ABB RAPID module: FOUNDRY.mod

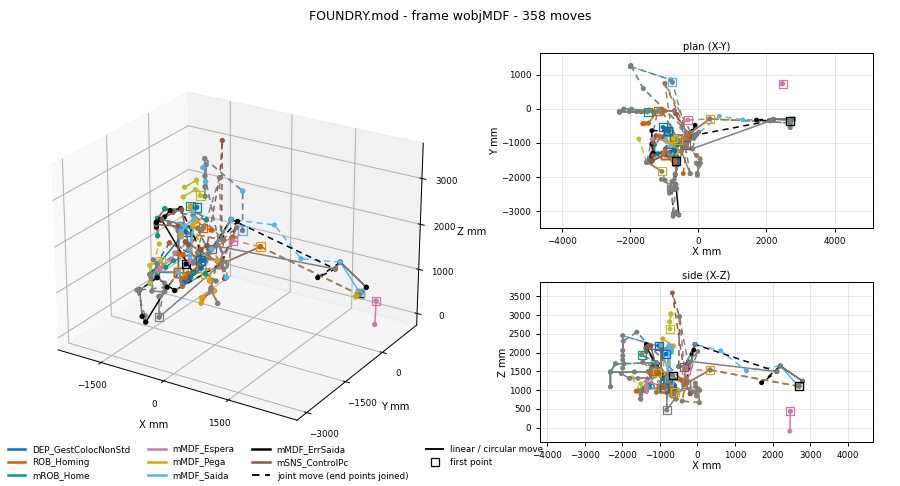
[picture p0: tool path of FOUNDRY.mod in frame wobjMDF, 358 of 371 moves have a stored position in this frame; points joined in program order, loops and branches not executed]
MODULE FOUNDRY

    !***********************************************************************************
    !*Project:   customer			: CIE Autocom (BR)
    !*           robot s/n			: 8156
    !*
    !*Robot:     Robot System		: IRC5 6.04.01.00
    !*           Robot NR.			: 109474
    !*           Robot Option		:
    !*           Robot Type			: IRB 6700-205/2.80
    !*           Robot Software		:
    !*           TP Language		: PORTUGUES
    !*
    !*Periferie: DCM type			: COLOSIO PFO2000
    !*           cooling device		: vasca (cliente)
    !*           photosensors		: SI (Ligado ao conrolador do robô)
    !*           conveyor belt		: SI
    !*           spraying			: NO
    !*           trimming press		: SI (collegata a controller robot)I
    !*
    !*Created:	 2017-02-17
    !*Author:    A.Roberti
    !*Company:   RELBO srl
    !*Modified:  Fabio Luiz dos Santos
    !*Translated to portuguese: Fabio Luiz dos Santos
    !*
    !*THIS MODULE MUST BE USED WITH "TEXT", "UTILITY" AND "WLDZONES" MODULES.
    !***********************************************************************************

    !============ Conferir posições abaixo ============
    CONST robtarget p01:=[[2473.51,738.92,438.42],[0.454099,0.457405,0.552238,0.528779],[1,0,0,1],[9E+09,9E+09,9E+09,9E+09,9E+09,9E+09]];
    CONST robtarget p02:=[[2460.24,732.08,-92.92],[0.449187,0.452046,0.556362,0.533242],[1,0,0,1],[9E+09,9E+09,9E+09,9E+09,9E+09,9E+09]];
    PERS robtarget pTemp:=[[2468.78,703.01,-92.8363],[0.452338,0.45528,0.553646,0.530647],[1,0,0,1],[9E+09,9E+09,9E+09,9E+09,9E+09,9E+09]];
    CONST robtarget p04:=[[2373.93,-299.91,1461.99],[0.596392,-6.67991E-05,0.802693,-2.09958E-05],[1,-1,-1,1],[9E+09,9E+09,9E+09,9E+09,9E+09,9E+09]];
    CONST robtarget p05:=[[2373.93,-299.91,1461.99],[0.596392,-6.67991E-05,0.802693,-2.09958E-05],[1,-1,-1,1],[9E+09,9E+09,9E+09,9E+09,9E+09,9E+09]];
    CONST robtarget p06:=[[2373.93,-299.91,1461.99],[0.596392,-6.67991E-05,0.802693,-2.09958E-05],[1,-1,-1,1],[9E+09,9E+09,9E+09,9E+09,9E+09,9E+09]];
    CONST robtarget MDF_pRecog10:=[[2695.82,-242.69,1199.03],[0.998237,-0.00496931,0.0559359,-0.0192193],[1,-1,-1,1],[9E+09,9E+09,9E+09,9E+09,9E+09,9E+09]];

    CONST robtarget MDF_p23:=[[-309.29,-759.88,1174.58],[0.243259,-0.675086,-0.655856,-0.234385],[0,-1,0,0],[9E+09,9E+09,9E+09,9E+09,9E+09,9E+09]];
    CONST robtarget MDF_p41:=[[2057.65,-246.89,1441.09],[0.616132,-0.00865147,0.787526,0.0104616],[1,-1,0,1],[9E+09,9E+09,9E+09,9E+09,9E+09,9E+09]];
    CONST robtarget MDF_p40:=[[1706.22,-328.45,1196.02],[0.687339,-0.0878871,0.720939,-0.00939877],[1,-1,-1,1],[9E+09,9E+09,9E+09,9E+09,9E+09,9E+09]];
    CONST robtarget MDF_p51:=[[2695.80,-284.56,1199.03],[0.998236,-0.0049758,0.0559417,-0.0192583],[1,-1,-1,1],[9E+09,9E+09,9E+09,9E+09,9E+09,9E+09]];
    CONST robtarget MDF_p50:=[[2695.80,-284.56,1199.03],[0.998236,-0.00497575,0.0559413,-0.0192576],[1,-1,-1,1],[9E+09,9E+09,9E+09,9E+09,9E+09,9E+09]];
    CONST robtarget MDF_p60:=[[2695.80,-284.56,1199.03],[0.998236,-0.00497576,0.0559417,-0.0192575],[1,-1,-1,1],[9E+09,9E+09,9E+09,9E+09,9E+09,9E+09]];
    CONST robtarget MDF_p61:=[[2695.80,-284.56,1199.03],[0.998236,-0.00497571,0.0559408,-0.0192572],[1,-1,-1,1],[9E+09,9E+09,9E+09,9E+09,9E+09,9E+09]];
    CONST robtarget MDF_p22:=[[1102.79,-218.74,1895.07],[0.935496,-0.0143034,0.351181,0.036262],[1,-1,0,1],[9E+09,9E+09,9E+09,9E+09,9E+09,9E+09]];

    CONST robtarget MDF_p70:=[[93.40,-478.70,2065.31],[0.934668,0.0189998,0.0567069,-0.350456],[1,-1,0,1],[9E+09,9E+09,9E+09,9E+09,9E+09,9E+09]];
    CONST robtarget MDF_p71:=[[-94.08,-478.58,2065.27],[0.849875,0.0295531,0.0520109,-0.523578],[0,-1,0,1],[9E+09,9E+09,9E+09,9E+09,9E+09,9E+09]];
    CONST robtarget MDF_p80:=[[1370.80,-212.89,1499.22],[0.814032,-0.0190361,0.57994,0.0256936],[1,-1,-1,1],[9E+09,9E+09,9E+09,9E+09,9E+09,9E+09]];
    CONST robtarget MDF_p81:=[[1306.48,-320.84,1511.93],[0.617506,-0.130992,0.771355,0.0808671],[1,-1,0,1],[9E+09,9E+09,9E+09,9E+09,9E+09,9E+09]];

    CONST robtarget MDF_p91:=[[617.59,-214.31,2051.16],[0.805845,-0.0646225,-0.0933712,0.581137],[1,0,0,1],[9E+09,9E+09,9E+09,9E+09,9E+09,9E+09]];
    CONST robtarget MDF_p33:=[[319.27,-312.34,1536.54],[0.13049,0.0260758,0.991098,-0.00401919],[1,-1,0,0],[9E+09,9E+09,9E+09,9E+09,9E+09,9E+09]];
    CONST robtarget MDF_pControl10:=[[448.88,-592.67,2016.31],[0.996524,0.0429781,0.0652434,-0.0289314],[1,0,0,1],[9E+09,9E+09,9E+09,9E+09,9E+09,9E+09]];
    CONST robtarget MDF_p43:=[[2697.36,-501.35,1107.86],[0.998235,-0.00496071,0.055963,-0.0192532],[1,-1,0,1],[9E+09,9E+09,9E+09,9E+09,9E+09,9E+09]];
    CONST robtarget MDF_p32:=[[-148.76,-493.05,1985.25],[0.747821,0.0411262,0.131836,-0.649378],[0,-1,-1,1],[9E+09,9E+09,9E+09,9E+09,9E+09,9E+09]];
    CONST robtarget SNS_p21:=[[-309.29,-759.88,1174.58],[0.243257,-0.67509,-0.655856,-0.234378],[0,-1,0,0],[9E+09,9E+09,9E+09,9E+09,9E+09,9E+09]];
    CONST robtarget pControl_01:=[[-304.77,-1154.52,1895.14],[0.698253,-0.00430576,0.705523,-0.121086],[0,-2,0,1],[9E+09,9E+09,9E+09,9E+09,9E+09,9E+09]];


    !===================================================================================
    ! EIXOS EM 0 GRAUS PARA VERIFICAR CALIBRACAO
    CONST jointtarget jposCalib:=[[0.0,0.0,0.0,0.0,0.0,0.0],[9E+09,9E+09,9E+09,9E+09,9E+09,9E+09]];
    ! POSICAO DE TRANSPORTE
    CONST jointtarget jposTransporte:=[[0.00449267,-45.002,64.9985,0.000647968,-115.001,4.99587],[9E+09,9E+09,9E+09,9E+09,9E+09,9E+09]];
    !===================================================================================
    ! HOME POSICAO (POSICAO INICIAL)
    CONST robtarget ROB_pHome:=[[-309.29,-759.88,1174.59],[0.243259,-0.67509,-0.655854,-0.23438],[0,-1,0,0],[9E+09,9E+09,9E+09,9E+09,9E+09,9E+09]];
    !===================================================================================
    ! M?QUINA DE FUNDICAO (MDF): ESPERA
    CONST robtarget MDF_pEspera:=[[335.19,-295.19,1536.55],[0.13056,9.64202E-05,0.99144,-0.00060735],[1,-1,0,0],[9E+09,9E+09,9E+09,9E+09,9E+09,9E+09]];
    !===================================================================================
    ! MAQUINA DE FUNDICAO (MDF): ENTRADA
    CONST robtarget MDF_p01:=[[2704.71,-411.78,1100.79],[0.587037,0.011242,0.809463,0.00555487],[1,-1,0,1],[9E+09,9E+09,9E+09,9E+09,9E+09,9E+09]];
    CONST robtarget MDF_p02:=[[2697.36,-357.61,1107.87],[0.998235,-0.00496108,0.0559633,-0.0192572],[1,-1,-1,1],[9E+09,9E+09,9E+09,9E+09,9E+09,9E+09]];
    CONST robtarget MDF_p03:=[[2697.37,-358.92,1107.86],[0.998235,-0.00495896,0.0559656,-0.0192394],[1,-1,-1,1],[9E+09,9E+09,9E+09,9E+09,9E+09,9E+09]];
    CONST robtarget MDF_pPega:=[[2697.36,-549.12,1107.87],[0.998235,-0.00496031,0.055963,-0.0192579],[1,-1,0,1],[9E+09,9E+09,9E+09,9E+09,9E+09,9E+09]];
    PERS robtarget MDF_pTemp:=[[2694.21,-536.375,1106.5],[0.998116,-0.00503237,0.0568545,-0.0225023],[1,-1,0,1],[9E+09,9E+09,9E+09,9E+09,9E+09,9E+09]];
    CONST robtarget MDF_p04:=[[2697.36,-297.72,1107.87],[0.998235,-0.00496111,0.0559628,-0.019259],[1,-1,-1,1],[9E+09,9E+09,9E+09,9E+09,9E+09,9E+09]];
    !===================================================================================
    ! MAQUINA DE FUNDICAO (MDF): SALIDA
    CONST robtarget MDF_p10:=[[2798.70,-298.15,1239.60],[0.868299,-0.0143122,0.495492,-0.0184121],[1,-1,-1,1],[9E+09,9E+09,9E+09,9E+09,9E+09,9E+09]];
    CONST robtarget MDF_p11:=[[2203.10,-303.56,1644.90],[0.856797,-0.177507,0.433581,0.215401],[1,-1,0,1],[9E+09,9E+09,9E+09,9E+09,9E+09,9E+09]];
    CONST robtarget MDF_p12:=[[2114.45,-349.91,1492.71],[0.599346,-0.117299,0.78976,0.0574839],[1,-1,0,1],[9E+09,9E+09,9E+09,9E+09,9E+09,9E+09]];
    CONST robtarget MDF_p20:=[[1642.01,-439.61,1289.54],[0.823576,-5.9409E-05,0.567206,-1.43407E-05],[1,-1,0,1],[9E+09,9E+09,9E+09,9E+09,9E+09,9E+09]];
    CONST robtarget MDF_p21:=[[992.58,-330.88,1566.27],[0.702618,-0.0208979,0.710504,-0.0327757],[1,-1,0,1],[9E+09,9E+09,9E+09,9E+09,9E+09,9E+09]];
    CONST robtarget MDF_pControl:=[[-165.98,-1166.57,1763.98],[0.60515,0.0268408,0.791448,-0.0817503],[0,-2,0,1],[9E+09,9E+09,9E+09,9E+09,9E+09,9E+09]];
    CONST robtarget MDF_pControl_11:=[[-304.77,-1154.52,1895.14],[0.698253,-0.00430576,0.705523,-0.121086],[0,-2,0,1],[9E+09,9E+09,9E+09,9E+09,9E+09,9E+09]];
    CONST robtarget MDF_p30:=[[-66.69,-765.21,2217.81],[0.991581,-0.108659,-0.0385252,-0.0589544],[0,0,0,1],[9E+09,9E+09,9E+09,9E+09,9E+09,9E+09]];
    CONST robtarget MDF_p31:=[[-350.61,-1056.76,1612.90],[0.680926,0.0158107,0.727045,-0.0865753],[-1,-2,0,1],[9E+09,9E+09,9E+09,9E+09,9E+09,9E+09]];
    CONST robtarget MDF_p13:=[[-309.29,-759.89,1174.59],[0.243258,-0.67509,-0.655855,-0.23438],[0,-1,0,0],[9E+09,9E+09,9E+09,9E+09,9E+09,9E+09]];
    CONST robtarget MDF_p14:=[[12.02,-682.53,2028.46],[0.998079,0.0593523,0.0134589,-0.0115613],[0,-1,0,1],[9E+09,9E+09,9E+09,9E+09,9E+09,9E+09]];
    !===================================================================================
    ! SENSORES
    CONST robtarget SNS_p01:=[[-350.61,-1056.76,1612.89],[0.680927,0.0158161,0.727044,-0.0865756],[-1,-2,0,1],[9E+09,9E+09,9E+09,9E+09,9E+09,9E+09]];
    CONST robtarget SNS_p02:=[[-498.09,-998.45,1630.02],[0.680911,0.0157817,0.727055,-0.086622],[-1,-2,0,1],[9E+09,9E+09,9E+09,9E+09,9E+09,9E+09]];
    CONST robtarget SNS_pControl1:=[[-498.07,-1238.79,1630.02],[0.680913,0.0157813,0.727053,-0.0866156],[-1,-2,0,1],[9E+09,9E+09,9E+09,9E+09,9E+09,9E+09]];
    CONST robtarget SNS_pControl2:=[[-236.59,-1901.29,1658.69],[0.555085,0.419469,-0.460857,0.550942],[0,1,0,0],[9E+09,9E+09,9E+09,9E+09,9E+09,9E+09]];
    CONST robtarget SNS_pControl3:=[[-236.59,-1901.29,1658.69],[0.555086,0.419469,-0.460856,0.550942],[0,1,0,0],[9E+09,9E+09,9E+09,9E+09,9E+09,9E+09]];
    CONST robtarget SNS_pControl4:=[[-236.59,-1901.29,1658.69],[0.555085,0.419469,-0.460857,0.550942],[0,1,0,0],[9E+09,9E+09,9E+09,9E+09,9E+09,9E+09]];
    CONST robtarget SNS_p10:=[[-479.84,-542.93,2956.94],[0.0253695,-0.0230724,0.928121,-0.370697],[-1,-2,0,1],[9E+09,9E+09,9E+09,9E+09,9E+09,9E+09]];
    CONST robtarget SNS_p11:=[[-309.29,-759.88,1174.59],[0.24326,-0.67509,-0.655854,-0.234381],[0,-1,0,0],[9E+09,9E+09,9E+09,9E+09,9E+09,9E+09]];
    !=====================================================================================
    ! CUBA DE AGUA
    CONST robtarget ENF_p01:=[[-816.23,-2285.86,928.08],[0.215617,0.952924,0.0580622,0.205121],[0,0,0,0],[9E+09,9E+09,9E+09,9E+09,9E+09,9E+09]];
    CONST robtarget ENF_p02:=[[-440.63,-1897.38,1282.18],[0.718138,0.0885909,0.689911,-0.0212891],[0,-2,0,1],[9E+09,9E+09,9E+09,9E+09,9E+09,9E+09]];
    CONST robtarget ENF_p03:=[[-573.40,-2628.84,1240.28],[0.718462,0.0885711,0.689567,-0.0215669],[0,-2,0,1],[9E+09,9E+09,9E+09,9E+09,9E+09,9E+09]];
    CONST robtarget ENF_p04:=[[-785.25,-1953.16,845.96],[0.631902,0.761096,0.0876551,0.11726],[0,1,-1,0],[9E+09,9E+09,9E+09,9E+09,9E+09,9E+09]];
    CONST robtarget ENF_pCuba:=[[-816.30,-2285.83,472.77],[0.215579,0.952925,0.0580234,0.205164],[0,0,0,0],[9E+09,9E+09,9E+09,9E+09,9E+09,9E+09]];
    CONST robtarget ENF_p10:=[[-778.88,-2131.13,1173.74],[0.71674,0.696411,0.000326903,-0.0360001],[0,1,-1,0],[9E+09,9E+09,9E+09,9E+09,9E+09,9E+09]];
    CONST robtarget ENF_p11:=[[-780.71,-2290.62,948.87],[0.631901,0.761095,0.0876729,0.117254],[0,1,-1,0],[9E+09,9E+09,9E+09,9E+09,9E+09,9E+09]];
    CONST robtarget ENF_p12:=[[29.47,-1884.57,501.58],[0.106643,-0.639134,-0.750945,0.127342],[0,-3,2,1],[9E+09,9E+09,9E+09,9E+09,9E+09,9E+09]];
    CONST robtarget ENF_p20:=[[-633.19,-2343.32,1104.45],[0.431426,0.658438,-0.391718,0.476328],[0,1,0,0],[9E+09,9E+09,9E+09,9E+09,9E+09,9E+09]];
    CONST robtarget ENF_p21:=[[-1085.76,-2068.67,1587.93],[0.646248,0.686559,0.136448,-0.303944],[0,1,-2,0],[9E+09,9E+09,9E+09,9E+09,9E+09,9E+09]];
    CONST robtarget ENF_p22:=[[-972.77,-2097.81,1535.68],[0.696167,0.699868,-0.0129623,-0.159272],[0,1,-1,0],[9E+09,9E+09,9E+09,9E+09,9E+09,9E+09]];
    CONST robtarget ENF_p23:=[[-440.54,-1897.37,1282.17],[0.718139,0.0885822,0.689911,-0.0212782],[0,-2,0,1],[9E+09,9E+09,9E+09,9E+09,9E+09,9E+09]];
    !===================================================================================
    ! COLOCACAO PECA NO INTERMEDIARIO
    CONST robtarget UTL_p01:=[[-1070.06,-1835.10,1470.49],[0.466574,0.842745,-0.106745,-0.246362],[0,1,-1,1],[9E+09,9E+09,9E+09,9E+09,9E+09,9E+09]];
    CONST robtarget UTL_p02:=[[-1293.78,-1608.42,1558.93],[0.831149,0.370293,-0.213137,-0.355874],[0,0,0,1],[9E+09,9E+09,9E+09,9E+09,9E+09,9E+09]];
    CONST robtarget UTL_p03:=[[-1482.11,-1589.62,1388.74],[0.54708,0.552185,-0.433217,-0.456201],[0,0,0,1],[9E+09,9E+09,9E+09,9E+09,9E+09,9E+09]];
    CONST robtarget UTL_p04:=[[-1505.03,-1545.60,877.79],[0.493718,0.499244,-0.496928,-0.509962],[0,0,0,1],[9E+09,9E+09,9E+09,9E+09,9E+09,9E+09]];
    CONST robtarget UTL_pColoc:=[[-1509.62,-1576.07,771.05],[0.59829,0.613623,-0.36049,-0.368189],[0,0,0,1],[9E+09,9E+09,9E+09,9E+09,9E+09,9E+09]];
    CONST robtarget UTL_p10:=[[-1504.86,-1545.34,953.20],[0.493701,0.499248,-0.496933,-0.509969],[0,0,0,1],[9E+09,9E+09,9E+09,9E+09,9E+09,9E+09]];
    CONST robtarget UTL_p11:=[[-1742.50,-882.65,1329.94],[0.547038,0.552222,-0.433233,-0.45619],[-1,0,0,1],[9E+09,9E+09,9E+09,9E+09,9E+09,9E+09]];
    CONST robtarget UTL_p12:=[[-1479.96,-1594.74,1007.69],[0.547037,0.552216,-0.433221,-0.45621],[0,0,0,1],[9E+09,9E+09,9E+09,9E+09,9E+09,9E+09]];
    !===================================================================================
    ! RETIRADA PECA DO INTERMEDIARIO
    CONST robtarget UTL_p51:=[[-837.41,-1272.63,1959.31],[0.955925,0.0359635,-0.0135944,-0.291083],[0,0,0,1],[9E+09,9E+09,9E+09,9E+09,9E+09,9E+09]];
    CONST robtarget UTL_p52:=[[-1296.42,-1371.93,1145.58],[0.695048,0.651142,0.261802,0.156151],[-1,-2,1,1],[9E+09,9E+09,9E+09,9E+09,9E+09,9E+09]];
    CONST robtarget UTL_p53:=[[-1296.41,-1372.01,1145.58],[0.695055,0.651133,0.261809,0.156144],[-1,-2,1,1],[9E+09,9E+09,9E+09,9E+09,9E+09,9E+09]];
    CONST robtarget UTL_p54:=[[-1505.01,-1545.57,877.73],[0.493703,0.499257,-0.496926,-0.509965],[0,0,0,1],[9E+09,9E+09,9E+09,9E+09,9E+09,9E+09]];
    CONST robtarget UTL_pPega:=[[-1510.35,-1566.50,762.25],[0.502673,0.515186,-0.488253,-0.49347],[0,0,0,1],[9E+09,9E+09,9E+09,9E+09,9E+09,9E+09]];
    CONST robtarget UTL_p60:=[[-1504.87,-1545.36,953.30],[0.493713,0.499235,-0.496941,-0.509963],[0,0,0,1],[9E+09,9E+09,9E+09,9E+09,9E+09,9E+09]];
    CONST robtarget UTL_p61:=[[-1434.58,-1608.11,1694.89],[0.663,0.645996,-0.264879,-0.270111],[0,0,0,1],[9E+09,9E+09,9E+09,9E+09,9E+09,9E+09]];
    CONST robtarget UTL_p62:=[[-1196.41,-1319.01,1646.77],[0.655082,0.649295,-0.283991,-0.261979],[0,0,0,1],[9E+09,9E+09,9E+09,9E+09,9E+09,9E+09]];
    !===================================================================================
    ! PRENSA: COLOCACAO
    CONST robtarget PRN_p01:=[[-1193.80,-61.32,1513.33],[0.15952,0.928352,-0.262292,-0.20957],[-1,0,0,0],[9E+09,9E+09,9E+09,9E+09,9E+09,9E+09]];
    CONST robtarget PRN_p02:=[[-976.84,-61.28,1510.97],[0.233234,0.684208,-0.682248,-0.109542],[-1,0,0,0],[9E+09,9E+09,9E+09,9E+09,9E+09,9E+09]];
    CONST robtarget PRN_p03:=[[-1453.00,-37.75,1743.34],[0.498689,0.512749,-0.4968,-0.491515],[-1,0,0,1],[9E+09,9E+09,9E+09,9E+09,9E+09,9E+09]];
    CONST robtarget PRN_p04:=[[-2008.40,-78.87,1584.76],[0.505059,0.503661,-0.494129,-0.497069],[-1,0,0,1],[9E+09,9E+09,9E+09,9E+09,9E+09,9E+09]];
    CONST robtarget PRN_p05:=[[-2025.32,-80.39,1437.60],[0.519828,0.551911,-0.473982,-0.447788],[-1,-1,1,1],[9E+09,9E+09,9E+09,9E+09,9E+09,9E+09]];
    CONST robtarget PRN_p06:=[[-2012.84,-78.16,1221.12],[0.519832,0.551906,-0.47397,-0.447802],[-1,-1,1,1],[9E+09,9E+09,9E+09,9E+09,9E+09,9E+09]];
    PERS robtarget PRN_pColoc:=[[-2031.56,-75.53,1091.03],[0.510214,0.51944,-0.489066,-0.480291],[-1,-1,1,1],[9E+09,9E+09,9E+09,9E+09,9E+09,9E+09]];
    CONST robtarget PRN_p10:=[[-2025.32,-80.42,1437.60],[0.519832,0.551912,-0.473979,-0.447785],[-1,-1,1,1],[9E+09,9E+09,9E+09,9E+09,9E+09,9E+09]];
    CONST robtarget PRN_p11:=[[-1804.46,-79.94,1313.09],[0.501985,0.498001,-0.498114,-0.501885],[-1,0,0,1],[9E+09,9E+09,9E+09,9E+09,9E+09,9E+09]];
    CONST robtarget PRN_p12:=[[-1586.23,-73.82,1311.37],[0.501982,0.498008,-0.49812,-0.501876],[-1,0,0,1],[9E+09,9E+09,9E+09,9E+09,9E+09,9E+09]];
    CONST robtarget PRN_p13:=[[-695.62,-55.45,1352.81],[0.0390151,0.751501,-0.655563,0.0629308],[-1,0,0,0],[9E+09,9E+09,9E+09,9E+09,9E+09,9E+09]];
    CONST robtarget PRN_p14:=[[-695.62,-55.41,1352.84],[0.0390281,0.751508,-0.655556,0.0629139],[-1,0,0,0],[9E+09,9E+09,9E+09,9E+09,9E+09,9E+09]];
    !
    !   Posicoes de deposito na prensa dependentes de retirada da gaveta
    !
    PERS robtarget pDepositaPrensa_1:=[[-2031.56,-75.53,1091.03],[0.510214,0.51944,-0.489066,-0.480291],[-1,-1,1,1],[9E+09,9E+09,9E+09,9E+09,9E+09,9E+09]];
    PERS robtarget pDepositaPrensa_2:=[[-2025.94,-80.41,1132.31],[0.508364,0.51283,-0.495652,-0.482598],[-1,-1,1,1],[9E+09,9E+09,9E+09,9E+09,9E+09,9E+09]];
    PERS robtarget pDepositaPrensa_3:=[[-2032.75,-74.5,1096.36],[0.511914,0.521062,-0.487274,-0.478543],[-1,-1,1,1],[9E+09,9E+09,9E+09,9E+09,9E+09,9E+09]];
    PERS robtarget pDepositaPrensa_4:=[[-2029.34,-74.63,1090.39],[0.513337,0.522498,-0.485777,-0.476972],[-1,-1,1,1],[9E+09,9E+09,9E+09,9E+09,9E+09,9E+09]];
    PERS robtarget pDepositaPrensa_5:=[[-2022.17,-74.64,1099.64],[0.497093,0.506578,-0.50237,-0.493864],[-1,0,0,1],[9E+09,9E+09,9E+09,9E+09,9E+09,9E+09]];
    PERS robtarget pDepositaPrensa_6:=[[-2022.17,-74.64,1099.64],[0.497093,0.506578,-0.50237,-0.493864],[-1,0,0,1],[9E+09,9E+09,9E+09,9E+09,9E+09,9E+09]];
    !
    !===================================================================================
    ! PRENSA: RETIRADA
    CONST robtarget PRN_p50:=[[-1486.38,-85.78,1945.73],[0.0614075,-0.701391,-0.688555,0.173702],[-1,0,3,0],[9E+09,9E+09,9E+09,9E+09,9E+09,9E+09]];
    CONST robtarget PRN_p51:=[[-1089.99,-98.97,1732.92],[0.222555,0.667241,0.697434,0.137275],[-1,0,3,0],[9E+09,9E+09,9E+09,9E+09,9E+09,9E+09]];
    CONST robtarget PRN_p52:=[[-1959.35,-6.29,1703.73],[0.497499,-0.502459,-0.49938,0.500649],[-1,0,3,1],[9E+09,9E+09,9E+09,9E+09,9E+09,9E+09]];
    CONST robtarget PRN_p53:=[[-2182.85,-6.28,1702.88],[0.497495,-0.502467,-0.499382,0.500642],[-1,0,3,1],[9E+09,9E+09,9E+09,9E+09,9E+09,9E+09]];
    CONST robtarget PRN_p54:=[[-2317.52,-87.25,1480.78],[0.497056,-0.502836,-0.499704,0.500388],[-1,0,2,1],[9E+09,9E+09,9E+09,9E+09,9E+09,9E+09]];
    CONST robtarget PRN_pPega:=[[-2315.98,-96.83,1089.21],[0.490704,-0.516807,-0.502931,0.489061],[-1,0,2,1],[9E+09,9E+09,9E+09,9E+09,9E+09,9E+09]];
    CONST robtarget PRN_p60:=[[-2317.51,-87.34,1480.84],[0.497055,-0.502826,-0.499706,0.500396],[-1,0,2,1],[9E+09,9E+09,9E+09,9E+09,9E+09,9E+09]];
    PERS robtarget PRN_pTemp:=[[-2316.06,-93.5701,1089.29],[0.491053,-0.517111,-0.502528,0.488803],[-1,0,2,1],[9E+09,9E+09,9E+09,9E+09,9E+09,9E+09]];
    CONST robtarget PRN_p61:=[[-1678.54,-87.22,1484.07],[0.497052,-0.502829,-0.499705,0.500397],[-1,0,2,1],[9E+09,9E+09,9E+09,9E+09,9E+09,9E+09]];
    CONST robtarget PRN_p62:=[[-1311.96,-87.14,1489.51],[0.497048,-0.502826,-0.499714,0.500396],[-1,0,2,1],[9E+09,9E+09,9E+09,9E+09,9E+09,9E+09]];
    CONST robtarget PRN_p63:=[[-1092.13,-9.30,947.61],[0.0815013,0.703548,0.700857,0.0847224],[-1,-1,3,0],[9E+09,9E+09,9E+09,9E+09,9E+09,9E+09]];
    CONST robtarget PRN_p64:=[[-598.98,-913.23,947.59],[0.0319419,0.290082,0.949753,0.113141],[0,-1,3,0],[9E+09,9E+09,9E+09,9E+09,9E+09,9E+09]];
    !===================================================================================
    ! COLOCACAO PECAS PRENSADAS
    CONST robtarget PRD_p01:=[[-598.98,-913.22,947.58],[0.0319427,0.29008,0.949753,0.113145],[0,-1,3,0],[9E+09,9E+09,9E+09,9E+09,9E+09,9E+09]];
    CONST robtarget PRD_p02:=[[-50.71,-1363.97,1094.29],[0.00191503,-0.0234862,-0.999542,0.0190067],[0,-1,3,0],[9E+09,9E+09,9E+09,9E+09,9E+09,9E+09]];
    CONST robtarget PRD_p03:=[[-55.43,-1591.70,1187.18],[0.00354788,-0.0199922,-0.885811,0.463602],[0,-1,3,1],[9E+09,9E+09,9E+09,9E+09,9E+09,9E+09]];
    CONST robtarget PRD_p04:=[[58.64,-1591.72,996.45],[0.00917576,-0.0181044,-0.713176,0.700691],[0,0,3,1],[9E+09,9E+09,9E+09,9E+09,9E+09,9E+09]];
    CONST robtarget PRD_p05:=[[-30.44,-1889.60,941.82],[0.101591,0.134875,0.700168,-0.693724],[0,0,3,1],[9E+09,9E+09,9E+09,9E+09,9E+09,9E+09]];
    CONST robtarget PRD_pColoc:=[[-26.63,-1947.83,846.62],[0.101356,0.135188,0.70194,-0.691904],[0,0,3,1],[9E+09,9E+09,9E+09,9E+09,9E+09,9E+09]];
    CONST robtarget PRD_p10:=[[16.18,-1664.07,1038.80],[0.101612,0.134855,0.700166,-0.693727],[0,0,3,1],[9E+09,9E+09,9E+09,9E+09,9E+09,9E+09]];
    CONST robtarget PRD_p11:=[[52.63,-1466.45,665.43],[0.0494621,0.163348,0.969341,-0.176776],[0,0,3,1],[9E+09,9E+09,9E+09,9E+09,9E+09,9E+09]];
    CONST robtarget PRD_p12:=[[-406.21,-995.82,708.10],[0.0709997,-0.762183,-0.64124,-0.0533618],[0,-1,0,0],[9E+09,9E+09,9E+09,9E+09,9E+09,9E+09]];
    CONST robtarget PRD_p13:=[[-300.08,-925.37,1318.03],[0.134893,-0.694147,-0.694092,-0.134907],[0,0,-1,0],[9E+09,9E+09,9E+09,9E+09,9E+09,9E+09]];
    CONST robtarget PRD_p14:=[[-300.08,-925.36,1318.02],[0.134901,-0.694143,-0.694093,-0.134912],[0,-1,-1,0],[9E+09,9E+09,9E+09,9E+09,9E+09,9E+09]];
    !===================================================================================
    ! COLOCACAO PECAS BUENAS NO PRENSADAS
    CONST robtarget BUE_p01:=[[-759.39,780.44,1244.81],[0.0183214,0.397609,-0.916269,-0.0449719],[-2,0,0,0],[9E+09,9E+09,9E+09,9E+09,9E+09,9E+09]];
    CONST robtarget BUE_p02:=[[-801.96,852.75,2103.63],[0.0430726,0.395196,-0.91111,-0.108823],[-2,0,0,0],[9E+09,9E+09,9E+09,9E+09,9E+09,9E+09]];
    CONST robtarget BUE_p03:=[[-1988.80,1241.70,2449.23],[0.259679,0.259077,-0.593792,-0.71614],[-1,-1,1,0],[9E+09,9E+09,9E+09,9E+09,9E+09,9E+09]];
    CONST robtarget BUE_p04:=[[-1988.79,1241.69,2053.26],[0.259676,0.259086,-0.593799,-0.716132],[-1,-2,2,0],[9E+09,9E+09,9E+09,9E+09,9E+09,9E+09]];
    CONST robtarget BUE_p05:=[[-1988.76,1241.70,1805.81],[0.25967,0.259085,-0.593805,-0.71613],[-1,-2,2,0],[9E+09,9E+09,9E+09,9E+09,9E+09,9E+09]];
    CONST robtarget BUE_pColoc:=[[-1988.76,1241.69,1584.18],[0.259664,0.259098,-0.593815,-0.716119],[-1,-2,2,0],[9E+09,9E+09,9E+09,9E+09,9E+09,9E+09]];
    CONST robtarget BUE_p10:=[[-1985.91,1262.35,1916.04],[0.259663,0.259105,-0.593814,-0.716118],[-1,-2,2,0],[9E+09,9E+09,9E+09,9E+09,9E+09,9E+09]];
    CONST robtarget BUE_p11:=[[-1975.82,1272.45,2305.18],[0.259659,0.259098,-0.593821,-0.716116],[-1,-1,1,0],[9E+09,9E+09,9E+09,9E+09,9E+09,9E+09]];
    CONST robtarget BUE_p12:=[[-1614.06,595.84,2544.20],[0.658456,-0.346023,-0.57656,-0.338057],[-1,-1,2,0],[9E+09,9E+09,9E+09,9E+09,9E+09,9E+09]];
    CONST robtarget BUE_p13:=[[-126.73,-861.59,959.59],[0.204587,0.977405,-0.052988,-0.00400906],[0,0,0,0],[9E+09,9E+09,9E+09,9E+09,9E+09,9E+09]];
    CONST robtarget BUE_p14:=[[-979.16,747.62,1055.74],[0.131339,-0.551677,0.822506,0.043428],[-1,-1,1,0],[9E+09,9E+09,9E+09,9E+09,9E+09,9E+09]];
    !===================================================================================
    ! COLOCACAO PECAS RECHAZADAS: START-UP/RECHAZADA DE M?QUINA/INCOMPLETA
    CONST robtarget RCZ_p01:=[[-659.90,-1525.85,1389.57],[0.386144,0.482582,0.65385,-0.436449],[0,-1,0,1],[9E+09,9E+09,9E+09,9E+09,9E+09,9E+09]];
    CONST robtarget RCZ_p02:=[[-658.41,-2217.86,1145.62],[0.567372,0.77177,0.254549,-0.132907],[0,-1,1,1],[9E+09,9E+09,9E+09,9E+09,9E+09,9E+09]];
    CONST robtarget RCZ_p03:=[[-726.98,-3076.91,1411.38],[0.411636,0.447204,0.625299,-0.489454],[0,-2,0,1],[9E+09,9E+09,9E+09,9E+09,9E+09,9E+09]];
    CONST robtarget RCZ_p04:=[[-739.76,-3153.50,1435.03],[0.433312,0.412173,0.595657,-0.536234],[0,-2,0,1],[9E+09,9E+09,9E+09,9E+09,9E+09,9E+09]];
    CONST robtarget RCZ_p05:=[[-644.51,-3024.99,855.66],[0.623312,0.77459,0.0751147,0.0764888],[0,-2,2,1],[9E+09,9E+09,9E+09,9E+09,9E+09,9E+09]];
    CONST robtarget RCZ_pColoc:=[[-572.13,-3112.62,767.06],[0.642178,0.765469,-0.0243048,-0.0327572],[0,-2,2,1],[9E+09,9E+09,9E+09,9E+09,9E+09,9E+09]];
    CONST robtarget RCZ_p10:=[[-680.87,-3077.00,848.31],[0.657259,0.753612,0.00850808,0.00275107],[0,-2,2,1],[9E+09,9E+09,9E+09,9E+09,9E+09,9E+09]];
    CONST robtarget RCZ_p11:=[[-727.17,-3076.82,1411.41],[0.411594,0.447208,0.625315,-0.489465],[0,-2,0,1],[9E+09,9E+09,9E+09,9E+09,9E+09,9E+09]];
    CONST robtarget RCZ_p12:=[[-784.28,-2379.37,1387.75],[0.386131,0.482598,0.65385,-0.436443],[0,-1,0,1],[9E+09,9E+09,9E+09,9E+09,9E+09,9E+09]];
    CONST robtarget RCZ_p13:=[[-678.33,-1918.50,949.54],[0.292276,0.945872,0.0750043,-0.119479],[0,-1,0,0],[9E+09,9E+09,9E+09,9E+09,9E+09,9E+09]];
    CONST robtarget RCZ_p14:=[[-309.26,-759.84,1174.56],[0.243257,-0.675073,-0.655869,-0.23439],[0,-1,0,0],[9E+09,9E+09,9E+09,9E+09,9E+09,9E+09]];
    !=====================================================================================
    ! MONTAJE MOLDES
    CONST robtarget MMD_p01:=[[-192.77,-816.33,904.35],[0.00260453,0.707148,0.707053,0.00338157],[0,0,-1,0],[9E+09,9E+09,9E+09,9E+09,9E+09,9E+09]];
    CONST robtarget MMD_p02:=[[-192.77,-816.33,904.35],[0.00260554,0.707147,0.707054,0.00338055],[0,0,-1,0],[9E+09,9E+09,9E+09,9E+09,9E+09,9E+09]];
    !=====================================================================================
    ! POSICIONES PARA RECUPERACAO SEMI-AUTOMATICA DE LA POSICAO INICIAL
    VAR robtarget ROB_pStartHoming;
    VAR jointtarget ROB_jStartHoming;
    !===================================================================================
    VAR bool bErrCtrl1:=FALSE;
    VAR bool bErrCtrl2:=FALSE;
    VAR bool bErrCtrl3:=FALSE;
    VAR bool bErrCtrl4:=FALSE;
    VAR bool bAnomSnsPulver:=FALSE;
    VAR bool bErrCtrlSns:=FALSE;
    VAR bool bPcIncompleta:=FALSE;
    VAR bool bPcRejeicaoDeMdf:=FALSE;
    VAR bool bSnsDefect:=FALSE;
    VAR bool bPcBoaDeMdf:=FALSE;
    VAR bool bMassaloteKo:=FALSE;
    VAR bool bErrSnsPulver:=FALSE;
    VAR bool bInjecaoKo:=FALSE;
    VAR bool bPcColocada:=FALSE;
    VAR bool bErrSnsIntColoc:=FALSE;
    VAR bool bPrnOkColoc:=FALSE;
    VAR bool bPrnOkPega:=FALSE;
    VAR bool bPrnErrStart1:=FALSE;
    VAR bool bPrnErrStart2:=FALSE;
    VAR bool bQualidade:=FALSE;
    VAR bool bPegaCtrlMdf:=FALSE;
    !===================================================================================
    PERS num nSnsAusentes{10}:=[0,0,1,0,0,0,0,0,0,0];
    PERS num nSnsDefect{10}:=[0,0,0,0,0,0,0,0,0,0];
    VAR num ROB_nPosRobo;
    VAR num nMaxRobSpeed:=0;
    !===================================================================================
    VAR clock timerMDF;
    VAR clock timerEXT;
    VAR clock timerROB;
    !===================================================================================
    VAR intnum intQualidade:=0;
    VAR intnum intVel0:=0;
    VAR intnum intVelStd:=0;
    VAR intnum intMslKo:=0;
    !===================================================================================
    PERS bool bHbltcSnsAntPulver:=FALSE;
    PERS bool bHbltcSns01:=FALSE;
    PERS bool bHbltcSns02:=TRUE;
    PERS bool bHbltcSns03:=TRUE;
    PERS bool bHbltcSns04:=TRUE;
    PERS bool bHbltcSns05:=FALSE;
    PERS bool bHbltcSns06:=FALSE;
    PERS bool bHbltcSns07:=FALSE;
    PERS bool bHbltcSns08:=FALSE;
    PERS bool bHbltcSns09:=FALSE;
    PERS bool bHbltcSns10:=FALSE;
    PERS bool bHbltcSns11:=FALSE;
    PERS bool bHbltcSns12:=FALSE;
    PERS bool bHbltcSns13:=FALSE;
    PERS bool bHbltcSns14:=FALSE;
    PERS bool bHbltcSns15:=FALSE;
    PERS bool bHbltcSns16:=FALSE;
    PERS bool bHbltcSoftservo:=TRUE;
    PERS bool bHbltcGuardarIncompl:=FALSE;
    PERS bool bHbltcEsfriamento:=TRUE;
    PERS bool bHbltcEnfriaRejeicao:=FALSE;
    PERS bool bHbltcUtilInt:=TRUE;
    PERS bool bHbltcSnsUtilInt:=TRUE;
    PERS bool bHbltcPrensaColoc:=TRUE;
    PERS bool bHbltcPrensaPega:=TRUE;
    PERS bool bHbltcPrnPegaSoft:=TRUE;
    PERS bool bHbltcStopPrensaNoAuto:=FALSE;
    PERS bool bHbltcStopUtilSns:=FALSE;
    PERS bool bHbltcCicloSpec:=TRUE;
    PERS bool bHbltcCtrlMoldeAberto:=TRUE;
    !
    VAR bool fRetiraGaveta := FALSE;
    VAR bool fDepositaGaveta := FALSE;
    !===================================================================================
    PERS num nHbltcMensajes:=2;
    PERS num nTipoPcNaPinca:=0;
    PERS num nPass:=1234;
    PERS num nTempoEsfriam:=3;
    PERS num nTempoGotejamento:=2;
    PERS num nTempoMaxDIPrnColoc:=4;
    PERS num nTempoMaxDIPrnPega:=4;
    PERS num nTempPulsoEsteira:=50;
    PERS num nTempoMaxDIAr:=2;
    PERS num nTempoMaxDIEyecAdel:=10;
    PERS num nTempoMaxDIPrnFimCiclo:=60;
    PERS num nTempoGarraFechar:=0.7;
    PERS num nTempoGarraAbrir:=0.7;
    PERS num nTempoMensAnom:=5;
    PERS num nVelMax:=2000;
    PERS num nOverVel:=100;
    PERS num ROB_ntimerMDF:=125.467;
    PERS num ROB_nTimerEXT:=0;
    PERS num ROB_nTimerROB:=63.46;
    PERS num ROB_nPcTotal:=225784;
    PERS num ROB_nPcBuona:=205183;
    PERS num ROB_nPcRejeicao:=20601;
    !
    VAR num nRetirouDaGaveta := 0;
    !===================================================================================
    PERS loaddata loadPeca:=[4,[0,-10,300],[1,0,0,0],0,0,0];
    !===================================================================================
    !           Variaveis para controle do resfriador
    !===================================================================================
    PERS num nTempoGaveta{6}:=[0,0,0,0,0,0];
    PERS bool fGavetaPronta{5}:=[FALSE,FALSE,FALSE,FALSE,FALSE];
    PERS num Gaveta;
    PERS num clkTempoGaveta{6}:=[0,0,0,0,0,0];
    !
    PERS bool fGavetaVazia{6}:=[FALSE,FALSE,FALSE,FALSE,FALSE,FALSE];

    !num nContador;
    !DI_R001_Gaveta_1
    !DI_R002_Gaveta_2
    !DI_R003_Gaveta_3
    !DI_R004_Gaveta_4
    !DI_R005_Gaveta_5
    !DI_R006_Gaveta_6

    PERS bool fCtrlGavetaVazia:=FALSE;
    PERS num nHistoricoGavetas{3}:=[1,2,6];
    !===================================================================================
    ! ANGULOS (EJE 1) LIMITES DE LOS DISPOSITIVOS PERIFERICOS
    CONST num njRampaMin:=-180;
    CONST num njRampaMax:=-90;
    CONST num njPrensaMin:=-90;
    CONST num njPrensaMax:=-30;
    CONST num njUtilMin:=-30;
    CONST num njUtilMax:=10;
    CONST num njCubaMin:=10;
    CONST num njCubaMax:=90;
    CONST num njMdfMin:=90;
    CONST num njMdfMax:=180;
    !===================================================================================
    CONST robtarget MDF_pPega10:=[[2695.82,-242.69,1199.03],[0.998237,-0.00496931,0.0559359,-0.0192193],[1,-1,-1,1],[9E+09,9E+09,9E+09,9E+09,9E+09,9E+09]];
    CONST robtarget ppreviocolocac:=[[-1505.07,-1545.58,765.14],[0.493726,0.499237,-0.496918,-0.50997],[0,0,0,1],[9E+09,9E+09,9E+09,9E+09,9E+09,9E+09]];
    CONST robtarget UTL_pColoc10:=[[-1495.71,-1583.56,764.56],[0.543625,0.560869,-0.427638,-0.454999],[0,0,0,1],[9E+09,9E+09,9E+09,9E+09,9E+09,9E+09]];
    CONST robtarget UTL_p21:=[[-1495.69,-1583.50,749.63],[0.543604,0.5609,-0.427622,-0.455],[0,0,0,1],[9E+09,9E+09,9E+09,9E+09,9E+09,9E+09]];
    CONST robtarget UTL_p64:=[[-1495.05,-1579.67,743.64],[0.505618,0.501122,-0.490396,-0.502732],[0,0,0,1],[9E+09,9E+09,9E+09,9E+09,9E+09,9E+09]];
    CONST robtarget UTL_p74:=[[-97.35,-1261.17,2063.25],[0.0101798,-0.000288689,0.610976,-0.791583],[0,-1,3,1],[9E+09,9E+09,9E+09,9E+09,9E+09,9E+09]];
    CONST robtarget PRD_pColoc10:=[[1.79,-2225.35,819.17],[0.0771116,0.096386,0.710322,-0.692969],[0,0,3,1],[9E+09,9E+09,9E+09,9E+09,9E+09,9E+09]];
    CONST robtarget ROB_pHome10:=[[-304.10,-777.14,1431.10],[0.0369415,-0.661671,-0.748009,-0.0361818],[0,-1,-1,0],[9E+09,9E+09,9E+09,9E+09,9E+09,9E+09]];
    CONST robtarget ROB_pHome20:=[[-310.41,-957.32,1307.40],[0.050306,-0.713482,-0.697746,-0.0395439],[0,-1,0,0],[9E+09,9E+09,9E+09,9E+09,9E+09,9E+09]];
    CONST robtarget RCZ_p24:=[[-309.29,-759.88,1174.58],[0.243257,-0.67509,-0.655855,-0.234381],[0,-1,0,0],[9E+09,9E+09,9E+09,9E+09,9E+09,9E+09]];
    CONST robtarget MDF_pEspera10:=[[-304.33,-326.91,1536.55],[0.0906149,0.71073,0.691242,-0.0940054],[0,-1,0,0],[9E+09,9E+09,9E+09,9E+09,9E+09,9E+09]];
    CONST robtarget MDF_pEsperaprevio:=[[-304.33,-326.91,1536.55],[0.0906156,0.71073,0.691241,-0.0940062],[0,-1,0,0],[9E+09,9E+09,9E+09,9E+09,9E+09,9E+09]];
    CONST robtarget RCZ_pColoc10:=[[-659.43,-3115.29,625.79],[0.639716,0.76213,-0.0675573,-0.0731942],[0,0,0,0],[9E+09,9E+09,9E+09,9E+09,9E+09,9E+09]];
    CONST robtarget UTL_p72:=[[-976.84,-61.36,1510.92],[0.233233,0.684246,-0.68221,-0.109546],[-1,0,0,0],[9E+09,9E+09,9E+09,9E+09,9E+09,9E+09]];
    CONST robtarget PRN_p15:=[[-2009.27,-76.41,1270.86],[0.504209,0.502563,-0.493847,-0.499318],[-1,2,-2,0],[9E+09,9E+09,9E+09,9E+09,9E+09,9E+09]];
    CONST robtarget UTL_p82:=[[-667.88,-855.82,1202.64],[0.313713,0.89558,-0.312553,-0.0428065],[0,0,0,0],[9E+09,9E+09,9E+09,9E+09,9E+09,9E+09]];
    CONST robtarget ENF_pCuba10:=[[-765.27,-2180.15,366.46],[0.70004,0.712249,0.0237051,0.0456512],[0,1,-1,0],[9E+09,9E+09,9E+09,9E+09,9E+09,9E+09]];
    CONST robtarget ROB_pHome30:=[[519.14,-306.19,1863.93],[0.990215,-0.0193778,0.138139,-0.00408639],[1,-1,0,1],[9E+09,9E+09,9E+09,9E+09,9E+09,9E+09]];
    CONST robtarget ENF_p30:=[[-849.70,-2477.95,1114.69],[0.550471,0.423196,0.638536,-0.331902],[0,1,-2,0],[9E+09,9E+09,9E+09,9E+09,9E+09,9E+09]];
    PERS robtarget HomeBoaColoc:=[[-1034.08,-542.12,2185.07],[0.335659,0.823838,-0.447559,-0.0911931],[-1,0,0,0],[9E+09,9E+09,9E+09,9E+09,9E+09,9E+09]];
    PERS robtarget pQuebraRebarba_00:=[[-1464.03,-418.73,983.03],[0.18504,0.680485,-0.708178,-0.0344188],[-1,0,1,0],[9E+09,9E+09,9E+09,9E+09,9E+09,9E+09]];
    PERS robtarget pQuebraRebarba_01:=[[-1577.79,-430.58,983.02],[0.185041,0.680489,-0.708173,-0.034419],[-1,0,1,0],[9E+09,9E+09,9E+09,9E+09,9E+09,9E+09]];
    PERS robtarget pQuebraRebarba_02:=[[-1625.91,-434.48,972.65],[0.217046,0.671487,-0.705518,-0.0651132],[-1,0,1,0],[9E+09,9E+09,9E+09,9E+09,9E+09,9E+09]];
    PERS robtarget pQuebraRebarba_03:=[[-1034.08,-542.12,2185.07],[0.335659,0.823838,-0.447559,-0.0911931],[-1,0,0,0],[9E+09,9E+09,9E+09,9E+09,9E+09,9E+09]];
    CONST robtarget SNS_p20:=[[-668.05,-140.14,3587.32],[0.487668,-0.205013,-0.407095,0.744596],[-1,-2,0,1],[9E+09,9E+09,9E+09,9E+09,9E+09,9E+09]];
    CONST robtarget pDepGaveta_1_1:=[[-887.83,-639.91,1066.32],[0.00200241,-0.903455,-0.428667,0.00306339],[0,-1,0,0],[9E+09,9E+09,9E+09,9E+09,9E+09,9E+09]];
    CONST robtarget pDepGaveta_1_11:=[[-887.83,-639.90,1299.67],[0.718477,0.694315,-0.039361,-0.0129874],[-1,1,-1,0],[9E+09,9E+09,9E+09,9E+09,9E+09,9E+09]];
    CONST robtarget pDepGaveta_1_21:=[[-612.28,-1051.68,1126.85],[0.71752,0.695289,-0.0138636,-0.0393256],[0,1,-1,0],[9E+09,9E+09,9E+09,9E+09,9E+09,9E+09]];
    CONST robtarget pDepGaveta_1_31:=[[-612.26,-1436.70,1078.08],[0.717526,0.695283,-0.0138581,-0.0393292],[0,1,-1,0],[9E+09,9E+09,9E+09,9E+09,9E+09,9E+09]];
    CONST robtarget pDepGaveta_1_41:=[[-612.26,-1491.41,1059.36],[0.71753,0.695278,-0.0138587,-0.0393387],[0,1,-1,0],[9E+09,9E+09,9E+09,9E+09,9E+09,9E+09]];
    CONST robtarget pDepGaveta_1_51:=[[-612.24,-1634.60,1059.35],[0.717527,0.695281,-0.0138553,-0.0393363],[0,1,-1,0],[9E+09,9E+09,9E+09,9E+09,9E+09,9E+09]];
    CONST robtarget pDepGaveta_1_61:=[[-689.98,-1634.60,1059.36],[0.71753,0.695277,-0.0138582,-0.0393362],[0,1,-1,0],[9E+09,9E+09,9E+09,9E+09,9E+09,9E+09]];
    CONST robtarget pDepGaveta_1_71:=[[-689.40,-1620.66,999.30],[0.71763,0.695227,-0.0253275,-0.0320195],[0,1,-1,0],[9E+09,9E+09,9E+09,9E+09,9E+09,9E+09]];
    CONST robtarget pDepGaveta_1_81:=[[-689.40,-1620.66,1058.84],[0.717633,0.695223,-0.0253276,-0.0320244],[0,1,-1,0],[9E+09,9E+09,9E+09,9E+09,9E+09,9E+09]];
    CONST robtarget pDepGaveta_1_91:=[[-689.43,-1220.74,1058.83],[0.717633,0.695223,-0.0253383,-0.0320325],[0,1,-1,0],[9E+09,9E+09,9E+09,9E+09,9E+09,9E+09]];
    CONST robtarget pDepGaveta_1_101:=[[-887.83,-639.91,1066.32],[0.0020033,-0.903455,-0.428667,0.00306161],[0,-1,0,0],[9E+09,9E+09,9E+09,9E+09,9E+09,9E+09]];
    CONST robtarget pRetGaveta_1_1:=[[-689.40,-1620.65,1058.82],[0.717628,0.695229,-0.0253274,-0.0320226],[0,1,-1,0],[9E+09,9E+09,9E+09,9E+09,9E+09,9E+09]];
    CONST robtarget pRetGaveta_1_11:=[[-965.55,-1348.17,1058.82],[0.717628,0.695229,-0.0253369,-0.0320263],[-1,1,-1,0],[9E+09,9E+09,9E+09,9E+09,9E+09,9E+09]];
    CONST robtarget pRetGaveta_1_21:=[[-689.41,-1620.64,920.24],[0.717632,0.695225,-0.0253295,-0.0320307],[0,1,-1,0],[9E+09,9E+09,9E+09,9E+09,9E+09,9E+09]];
    CONST robtarget pRetGaveta_1_31:=[[-689.43,-1620.63,1063.70],[0.717629,0.695227,-0.025333,-0.0320299],[0,1,-1,0],[9E+09,9E+09,9E+09,9E+09,9E+09,9E+09]];
    CONST robtarget pRetGaveta_1_41:=[[-689.45,-1546.94,1063.70],[0.717632,0.695224,-0.0253349,-0.0320324],[0,1,-1,0],[9E+09,9E+09,9E+09,9E+09,9E+09,9E+09]];
    CONST robtarget pRetGaveta_1_51:=[[-689.45,-1546.94,1107.17],[0.717633,0.695223,-0.0253351,-0.0320331],[0,1,-1,0],[9E+09,9E+09,9E+09,9E+09,9E+09,9E+09]];
    CONST robtarget pRetGaveta_1_61:=[[-689.47,-1420.87,1107.16],[0.717632,0.695224,-0.0253434,-0.0320327],[0,1,-1,0],[9E+09,9E+09,9E+09,9E+09,9E+09,9E+09]];
    CONST robtarget pRetGaveta_1_71:=[[-689.48,-1420.86,1127.23],[0.717633,0.695223,-0.0253452,-0.0320365],[0,1,-1,0],[9E+09,9E+09,9E+09,9E+09,9E+09,9E+09]];
    CONST robtarget pRetGaveta_1_81:=[[-689.48,-998.43,1127.23],[0.717631,0.695224,-0.0253476,-0.032036],[-1,1,-1,0],[9E+09,9E+09,9E+09,9E+09,9E+09,9E+09]];
    CONST robtarget pRetGaveta_1_91:=[[-1148.72,-802.12,1488.02],[0.157725,-0.703899,-0.622036,-0.304501],[0,-1,-1,0],[9E+09,9E+09,9E+09,9E+09,9E+09,9E+09]];
    CONST robtarget pRetGaveta_1_101:=[[-309.29,-759.88,1174.59],[0.243259,-0.67509,-0.655853,-0.234381],[0,-1,0,0],[9E+09,9E+09,9E+09,9E+09,9E+09,9E+09]];
    !
    CONST robtarget pDepGaveta_2_1:=[[-887.83,-639.91,1066.32],[0.00200241,-0.903455,-0.428667,0.00306339],[0,-1,0,0],[9E+09,9E+09,9E+09,9E+09,9E+09,9E+09]];
    CONST robtarget pDepGaveta_2_11:=[[-887.83,-639.90,1299.67],[0.718477,0.694315,-0.039361,-0.0129874],[-1,1,-1,0],[9E+09,9E+09,9E+09,9E+09,9E+09,9E+09]];
    CONST robtarget pDepGaveta_2_21:=[[-1279.29,-1051.61,1126.86],[0.717519,0.695289,-0.0138761,-0.0393468],[-1,1,-1,0],[9E+09,9E+09,9E+09,9E+09,9E+09,9E+09]];
    CONST robtarget pDepGaveta_2_31:=[[-1279.23,-1342.85,1091.94],[0.718486,0.694312,-0.0391893,-0.013147],[-1,1,-1,0],[9E+09,9E+09,9E+09,9E+09,9E+09,9E+09]];
    CONST robtarget pDepGaveta_2_41:=[[-1410.30,-1473.63,1060.65],[0.718495,0.694303,-0.0391933,-0.0131524],[-1,1,-1,0],[9E+09,9E+09,9E+09,9E+09,9E+09,9E+09]];
    CONST robtarget pDepGaveta_2_51:=[[-1365.53,-1514.20,1024.95],[0.717783,0.695166,-0.0190546,-0.0341825],[-1,1,-1,0],[9E+09,9E+09,9E+09,9E+09,9E+09,9E+09]];
    CONST robtarget pDepGaveta_2_61:=[[-1363.62,-1521.64,996.70],[0.718023,0.695004,-0.0240115,-0.0288983],[-1,1,-1,0],[9E+09,9E+09,9E+09,9E+09,9E+09,9E+09]];
    CONST robtarget pDepGaveta_2_71:=[[-1363.63,-1521.62,966.07],[0.718023,0.695004,-0.0240179,-0.0288983],[-1,1,-1,0],[9E+09,9E+09,9E+09,9E+09,9E+09,9E+09]];
    CONST robtarget pDepGaveta_2_81:=[[-1363.63,-1521.62,1032.80],[0.718019,0.695008,-0.0240164,-0.028895],[-1,1,-1,0],[9E+09,9E+09,9E+09,9E+09,9E+09,9E+09]];
    CONST robtarget pDepGaveta_2_91:=[[-689.43,-1220.74,1058.83],[0.717633,0.695223,-0.0253383,-0.0320325],[0,1,-1,0],[9E+09,9E+09,9E+09,9E+09,9E+09,9E+09]];
    CONST robtarget pDepGaveta_2_101:=[[-887.83,-639.91,1066.32],[0.0020033,-0.903455,-0.428667,0.00306161],[0,-1,0,0],[9E+09,9E+09,9E+09,9E+09,9E+09,9E+09]];
    CONST robtarget pRetGaveta_2_1:=[[-1360.91,-1519.51,1059.96],[0.717614,0.695243,-0.0253454,-0.032009],[-1,1,-1,0],[9E+09,9E+09,9E+09,9E+09,9E+09,9E+09]];
    CONST robtarget pRetGaveta_2_11:=[[-965.55,-1348.17,1058.82],[0.717628,0.695229,-0.0253369,-0.0320263],[-1,1,-1,0],[9E+09,9E+09,9E+09,9E+09,9E+09,9E+09]];
    CONST robtarget pRetGaveta_2_21:=[[-1360.92,-1519.50,957.99],[0.717617,0.69524,-0.0253501,-0.0320121],[-1,1,-1,0],[9E+09,9E+09,9E+09,9E+09,9E+09,9E+09]];
    CONST robtarget pRetGaveta_2_31:=[[-1360.93,-1519.49,1073.36],[0.717611,0.695246,-0.025346,-0.0320143],[-1,1,-1,0],[9E+09,9E+09,9E+09,9E+09,9E+09,9E+09]];
    CONST robtarget pRetGaveta_2_41:=[[-1360.94,-1436.06,1073.36],[0.717613,0.695244,-0.0253507,-0.0320126],[-1,1,-1,0],[9E+09,9E+09,9E+09,9E+09,9E+09,9E+09]];
    CONST robtarget pRetGaveta_2_51:=[[-1357.30,-1298.28,1108.71],[0.717612,0.695245,-0.0253596,-0.0320175],[-1,1,-1,0],[9E+09,9E+09,9E+09,9E+09,9E+09,9E+09]];
    CONST robtarget pRetGaveta_2_61:=[[-1357.35,-1009.75,1119.51],[0.717609,0.695246,-0.0253776,-0.0320224],[-1,1,-1,0],[9E+09,9E+09,9E+09,9E+09,9E+09,9E+09]];
    CONST robtarget pRetGaveta_2_71:=[[-1357.35,-889.67,1222.23],[0.717607,0.695248,-0.0253809,-0.0320238],[-1,1,-1,0],[9E+09,9E+09,9E+09,9E+09,9E+09,9E+09]];
    CONST robtarget pRetGaveta_2_81:=[[-977.87,-915.06,1127.24],[0.717631,0.695222,-0.0253617,-0.0320579],[-1,1,-1,0],[9E+09,9E+09,9E+09,9E+09,9E+09,9E+09]];
    CONST robtarget pRetGaveta_2_91:=[[-1148.72,-802.12,1488.02],[0.157725,-0.703899,-0.622036,-0.304501],[0,-1,-1,0],[9E+09,9E+09,9E+09,9E+09,9E+09,9E+09]];
    CONST robtarget pRetGaveta_2_101:=[[-309.29,-759.88,1174.59],[0.243259,-0.67509,-0.655853,-0.234381],[0,-1,0,0],[9E+09,9E+09,9E+09,9E+09,9E+09,9E+09]];
    !
    CONST robtarget pDepGaveta_3_1:=[[-887.83,-639.91,1066.32],[0.00200241,-0.903455,-0.428667,0.00306339],[0,-1,0,0],[9E+09,9E+09,9E+09,9E+09,9E+09,9E+09]];
    CONST robtarget pDepGaveta_3_11:=[[-887.56,-632.59,1301.74],[0.715981,0.696197,-0.0037505,-0.0516536],[-1,1,-1,0],[9E+09,9E+09,9E+09,9E+09,9E+09,9E+09]];
    CONST robtarget pDepGaveta_3_21:=[[-922.80,-961.08,2367.18],[0.717513,0.695295,-0.0138566,-0.039345],[-1,0,0,0],[9E+09,9E+09,9E+09,9E+09,9E+09,9E+09]];
    CONST robtarget pDepGaveta_3_31:=[[-640.35,-1162.65,2179.28],[0.717513,0.695295,-0.0138555,-0.0393413],[0,0,0,0],[9E+09,9E+09,9E+09,9E+09,9E+09,9E+09]];
    CONST robtarget pDepGaveta_3_41:=[[-640.36,-1298.90,2169.04],[0.717515,0.695292,-0.0138425,-0.0393653],[0,0,0,0],[9E+09,9E+09,9E+09,9E+09,9E+09,9E+09]];
    CONST robtarget pDepGaveta_3_51:=[[-695.76,-1639.66,2051.60],[0.718722,0.694817,-0.0184441,-0.0180739],[0,0,0,0],[9E+09,9E+09,9E+09,9E+09,9E+09,9E+09]];
    CONST robtarget pDepGaveta_3_61:=[[-695.78,-1639.68,2097.48],[0.718709,0.694831,-0.0184472,-0.0180701],[0,0,0,0],[9E+09,9E+09,9E+09,9E+09,9E+09,9E+09]];
    CONST robtarget pDepGaveta_3_71:=[[-693.25,-1633.72,2063.86],[0.705615,0.708096,-0.00183369,-0.0265467],[0,0,0,0],[9E+09,9E+09,9E+09,9E+09,9E+09,9E+09]];
    CONST robtarget pDepGaveta_3_81:=[[-693.26,-1633.73,2127.98],[0.705608,0.708103,-0.00183266,-0.0265436],[0,0,0,0],[9E+09,9E+09,9E+09,9E+09,9E+09,9E+09]];
    CONST robtarget pDepGaveta_3_91:=[[-695.80,-1229.95,2097.50],[0.718709,0.694831,-0.018446,-0.0180894],[0,0,0,0],[9E+09,9E+09,9E+09,9E+09,9E+09,9E+09]];
    CONST robtarget pDepGaveta_3_101:=[[-887.83,-639.91,1066.32],[0.0020033,-0.903455,-0.428667,0.00306161],[0,-1,0,0],[9E+09,9E+09,9E+09,9E+09,9E+09,9E+09]];
    CONST robtarget pRetGaveta_3_1:=[[-973.16,-1258.37,2096.72],[0.717627,0.695229,-0.0253333,-0.0320295],[-1,0,0,0],[9E+09,9E+09,9E+09,9E+09,9E+09,9E+09]];
    CONST robtarget pRetGaveta_3_11:=[[-965.55,-1348.17,1058.82],[0.717628,0.695229,-0.0253369,-0.0320263],[-1,1,-1,0],[9E+09,9E+09,9E+09,9E+09,9E+09,9E+09]];
    CONST robtarget pRetGaveta_3_21:=[[-692.01,-1637.82,2013.79],[0.717802,0.695072,-0.0292244,-0.0279618],[0,0,0,0],[9E+09,9E+09,9E+09,9E+09,9E+09,9E+09]];
    CONST robtarget pRetGaveta_3_31:=[[-691.96,-1637.85,2139.28],[0.717799,0.695076,-0.0292108,-0.0279444],[0,0,0,0],[9E+09,9E+09,9E+09,9E+09,9E+09,9E+09]];
    CONST robtarget pRetGaveta_3_41:=[[-768.72,-1399.80,2139.28],[0.7178,0.695074,-0.0292222,-0.027947],[0,0,0,0],[9E+09,9E+09,9E+09,9E+09,9E+09,9E+09]];
    CONST robtarget pRetGaveta_3_51:=[[-758.48,-1058.65,2195.84],[0.717802,0.695072,-0.0292374,-0.0279391],[-1,0,0,0],[9E+09,9E+09,9E+09,9E+09,9E+09,9E+09]];
    CONST robtarget pRetGaveta_3_61:=[[-689.47,-1420.87,1107.16],[0.717632,0.695224,-0.0253434,-0.0320327],[0,1,-1,0],[9E+09,9E+09,9E+09,9E+09,9E+09,9E+09]];
    CONST robtarget pRetGaveta_3_71:=[[-964.49,-792.44,2195.84],[0.717806,0.695067,-0.0292549,-0.0279501],[-1,0,0,0],[9E+09,9E+09,9E+09,9E+09,9E+09,9E+09]];
    CONST robtarget pRetGaveta_3_81:=[[-962.13,-867.85,1127.23],[0.717632,0.695223,-0.0253519,-0.0320444],[-1,1,-1,0],[9E+09,9E+09,9E+09,9E+09,9E+09,9E+09]];
    CONST robtarget pRetGaveta_3_91:=[[-1148.72,-802.12,1488.02],[0.157725,-0.703899,-0.622036,-0.304501],[0,-1,-1,0],[9E+09,9E+09,9E+09,9E+09,9E+09,9E+09]];
    CONST robtarget pRetGaveta_3_101:=[[-309.29,-759.88,1174.59],[0.243259,-0.67509,-0.655853,-0.234381],[0,-1,0,0],[9E+09,9E+09,9E+09,9E+09,9E+09,9E+09]];
    !
    CONST robtarget pDepGaveta_4_1:=[[-887.83,-639.91,1066.32],[0.00200241,-0.903455,-0.428667,0.00306339],[0,-1,0,0],[9E+09,9E+09,9E+09,9E+09,9E+09,9E+09]];
    CONST robtarget pDepGaveta_4_11:=[[-887.83,-639.90,1299.67],[0.718477,0.694315,-0.039361,-0.0129874],[-1,1,-1,0],[9E+09,9E+09,9E+09,9E+09,9E+09,9E+09]];
    CONST robtarget pDepGaveta_4_21:=[[-1364.02,-640.02,2121.36],[0.713203,0.699959,-0.0253897,-0.0274773],[-1,0,0,0],[9E+09,9E+09,9E+09,9E+09,9E+09,9E+09]];
    CONST robtarget pDepGaveta_4_31:=[[-1363.99,-1028.12,2216.45],[0.713196,0.699967,-0.0253812,-0.0274629],[-1,0,0,0],[9E+09,9E+09,9E+09,9E+09,9E+09,9E+09]];
    CONST robtarget pDepGaveta_4_41:=[[-1322.58,-1290.89,2179.30],[0.713191,0.699974,-0.0253663,-0.027433],[-1,0,0,0],[9E+09,9E+09,9E+09,9E+09,9E+09,9E+09]];
    CONST robtarget pDepGaveta_4_51:=[[-1362.30,-1383.62,2140.09],[0.712889,0.700428,-0.00886681,-0.0333328],[-1,0,0,0],[9E+09,9E+09,9E+09,9E+09,9E+09,9E+09]];
    CONST robtarget pDepGaveta_4_61:=[[-1362.30,-1383.61,2140.09],[0.712889,0.700428,-0.00886701,-0.0333343],[-1,0,0,0],[9E+09,9E+09,9E+09,9E+09,9E+09,9E+09]];
    CONST robtarget pDepGaveta_4_71:=[[-1362.28,-1526.99,2140.09],[0.712887,0.700431,-0.00886509,-0.0333277],[-1,0,0,0],[9E+09,9E+09,9E+09,9E+09,9E+09,9E+09]];
    CONST robtarget pDepGaveta_4_81:=[[-1362.28,-1526.99,2140.09],[0.712886,0.700431,-0.00886465,-0.0333284],[-1,0,0,0],[9E+09,9E+09,9E+09,9E+09,9E+09,9E+09]];
    CONST robtarget pDepGaveta_4_91:=[[-689.43,-1220.74,1058.83],[0.717633,0.695223,-0.0253383,-0.0320325],[0,1,-1,0],[9E+09,9E+09,9E+09,9E+09,9E+09,9E+09]];
    CONST robtarget pDepGaveta_4_101:=[[-887.83,-639.91,1066.32],[0.0020033,-0.903455,-0.428667,0.00306161],[0,-1,0,0],[9E+09,9E+09,9E+09,9E+09,9E+09,9E+09]];
    CONST robtarget pRetGaveta_4_1:=[[-965.55,-1348.17,2081.39],[0.717626,0.69523,-0.0253349,-0.032024],[-1,0,0,0],[9E+09,9E+09,9E+09,9E+09,9E+09,9E+09]];
    CONST robtarget pRetGaveta_4_11:=[[-965.55,-1348.17,1058.82],[0.717628,0.695229,-0.0253369,-0.0320263],[-1,1,-1,0],[9E+09,9E+09,9E+09,9E+09,9E+09,9E+09]];
    CONST robtarget pRetGaveta_4_21:=[[-1367.74,-1529.01,2020.71],[0.717632,0.695223,-0.0253428,-0.032035],[-1,0,0,0],[9E+09,9E+09,9E+09,9E+09,9E+09,9E+09]];
    CONST robtarget pRetGaveta_4_31:=[[-1367.75,-1529.02,2133.08],[0.71762,0.695236,-0.0253403,-0.0320232],[-1,0,0,0],[9E+09,9E+09,9E+09,9E+09,9E+09,9E+09]];
    CONST robtarget pRetGaveta_4_41:=[[-1332.28,-1370.32,2152.63],[0.717618,0.695239,-0.0253276,-0.0320218],[-1,0,0,0],[9E+09,9E+09,9E+09,9E+09,9E+09,9E+09]];
    CONST robtarget pRetGaveta_4_51:=[[-1315.31,-996.84,2174.64],[0.717631,0.695224,-0.0253383,-0.0320501],[-1,0,0,0],[9E+09,9E+09,9E+09,9E+09,9E+09,9E+09]];
    CONST robtarget pRetGaveta_4_61:=[[-1240.88,-790.07,2174.63],[0.717629,0.695225,-0.025345,-0.0320568],[-1,0,0,0],[9E+09,9E+09,9E+09,9E+09,9E+09,9E+09]];
    CONST robtarget pRetGaveta_4_71:=[[-1240.88,-790.07,2174.63],[0.717629,0.695226,-0.0253465,-0.0320574],[-1,0,0,0],[9E+09,9E+09,9E+09,9E+09,9E+09,9E+09]];
    CONST robtarget pRetGaveta_4_81:=[[-1063.15,-819.26,1450.76],[0.717626,0.695228,-0.0253612,-0.0320511],[-1,1,-1,0],[9E+09,9E+09,9E+09,9E+09,9E+09,9E+09]];
    CONST robtarget pRetGaveta_4_91:=[[-1148.72,-802.12,1488.02],[0.157725,-0.703899,-0.622036,-0.304501],[0,-1,-1,0],[9E+09,9E+09,9E+09,9E+09,9E+09,9E+09]];
    CONST robtarget pRetGaveta_4_101:=[[-309.29,-759.88,1174.59],[0.243259,-0.67509,-0.655853,-0.234381],[0,-1,0,0],[9E+09,9E+09,9E+09,9E+09,9E+09,9E+09]];
    !
    CONST robtarget pDepGaveta_5_1:=[[-887.83,-639.91,1066.32],[0.00200241,-0.903455,-0.428667,0.00306339],[0,-1,0,0],[9E+09,9E+09,9E+09,9E+09,9E+09,9E+09]];
    CONST robtarget pDepGaveta_5_11:=[[-887.83,-639.90,1299.67],[0.718477,0.694315,-0.039361,-0.0129874],[-1,1,-1,0],[9E+09,9E+09,9E+09,9E+09,9E+09,9E+09]];
    CONST robtarget pDepGaveta_5_21:=[[-612.28,-1051.68,1126.85],[0.71752,0.695289,-0.0138636,-0.0393256],[0,1,-1,0],[9E+09,9E+09,9E+09,9E+09,9E+09,9E+09]];
    CONST robtarget pDepGaveta_5_31:=[[-612.26,-1436.70,1078.08],[0.717526,0.695283,-0.0138581,-0.0393292],[0,1,-1,0],[9E+09,9E+09,9E+09,9E+09,9E+09,9E+09]];
    CONST robtarget pDepGaveta_5_41:=[[-612.26,-1491.41,1059.36],[0.71753,0.695278,-0.0138587,-0.0393387],[0,1,-1,0],[9E+09,9E+09,9E+09,9E+09,9E+09,9E+09]];
    CONST robtarget pDepGaveta_5_51:=[[-612.24,-1634.60,1059.35],[0.717527,0.695281,-0.0138553,-0.0393363],[0,1,-1,0],[9E+09,9E+09,9E+09,9E+09,9E+09,9E+09]];
    CONST robtarget pDepGaveta_5_61:=[[-689.98,-1634.60,1059.36],[0.71753,0.695277,-0.0138582,-0.0393362],[0,1,-1,0],[9E+09,9E+09,9E+09,9E+09,9E+09,9E+09]];
    CONST robtarget pDepGaveta_5_71:=[[-689.40,-1620.66,999.30],[0.71763,0.695227,-0.0253275,-0.0320195],[0,1,-1,0],[9E+09,9E+09,9E+09,9E+09,9E+09,9E+09]];
    CONST robtarget pDepGaveta_5_81:=[[-689.40,-1620.66,1058.84],[0.717633,0.695223,-0.0253276,-0.0320244],[0,1,-1,0],[9E+09,9E+09,9E+09,9E+09,9E+09,9E+09]];
    CONST robtarget pDepGaveta_5_91:=[[-689.43,-1220.74,1058.83],[0.717633,0.695223,-0.0253383,-0.0320325],[0,1,-1,0],[9E+09,9E+09,9E+09,9E+09,9E+09,9E+09]];
    CONST robtarget pDepGaveta_5_101:=[[-887.83,-639.91,1066.32],[0.0020033,-0.903455,-0.428667,0.00306161],[0,-1,0,0],[9E+09,9E+09,9E+09,9E+09,9E+09,9E+09]];
    CONST robtarget pRetGaveta_5_1:=[[-689.40,-1620.65,1058.82],[0.717628,0.695229,-0.0253274,-0.0320226],[0,1,-1,0],[9E+09,9E+09,9E+09,9E+09,9E+09,9E+09]];
    CONST robtarget pRetGaveta_5_11:=[[-965.55,-1348.17,1058.82],[0.717628,0.695229,-0.0253369,-0.0320263],[-1,1,-1,0],[9E+09,9E+09,9E+09,9E+09,9E+09,9E+09]];
    CONST robtarget pRetGaveta_5_21:=[[-689.41,-1620.64,945.25],[0.717631,0.695226,-0.0253295,-0.0320275],[0,1,-1,0],[9E+09,9E+09,9E+09,9E+09,9E+09,9E+09]];
    CONST robtarget pRetGaveta_5_31:=[[-689.43,-1620.63,1063.70],[0.717629,0.695227,-0.025333,-0.0320299],[0,1,-1,0],[9E+09,9E+09,9E+09,9E+09,9E+09,9E+09]];
    CONST robtarget pRetGaveta_5_41:=[[-689.45,-1546.94,1063.70],[0.717632,0.695224,-0.0253349,-0.0320324],[0,1,-1,0],[9E+09,9E+09,9E+09,9E+09,9E+09,9E+09]];
    CONST robtarget pRetGaveta_5_51:=[[-689.45,-1546.94,1107.17],[0.717633,0.695223,-0.0253351,-0.0320331],[0,1,-1,0],[9E+09,9E+09,9E+09,9E+09,9E+09,9E+09]];
    CONST robtarget pRetGaveta_5_61:=[[-689.47,-1420.87,1107.16],[0.717632,0.695224,-0.0253434,-0.0320327],[0,1,-1,0],[9E+09,9E+09,9E+09,9E+09,9E+09,9E+09]];
    CONST robtarget pRetGaveta_5_71:=[[-689.48,-1420.86,1127.23],[0.717633,0.695223,-0.0253452,-0.0320365],[0,1,-1,0],[9E+09,9E+09,9E+09,9E+09,9E+09,9E+09]];
    CONST robtarget pRetGaveta_5_81:=[[-689.48,-998.43,1127.23],[0.717631,0.695224,-0.0253476,-0.032036],[-1,1,-1,0],[9E+09,9E+09,9E+09,9E+09,9E+09,9E+09]];
    CONST robtarget pRetGaveta_5_91:=[[-1148.72,-802.12,1488.02],[0.157725,-0.703899,-0.622036,-0.304501],[0,-1,-1,0],[9E+09,9E+09,9E+09,9E+09,9E+09,9E+09]];
    CONST robtarget pRetGaveta_5_101:=[[-309.29,-759.88,1174.59],[0.243259,-0.67509,-0.655853,-0.234381],[0,-1,0,0],[9E+09,9E+09,9E+09,9E+09,9E+09,9E+09]];
    !
    CONST robtarget pDepGaveta_6_1:=[[-887.83,-639.91,1066.32],[0.00200241,-0.903455,-0.428667,0.00306339],[0,-1,0,0],[9E+09,9E+09,9E+09,9E+09,9E+09,9E+09]];
    CONST robtarget pDepGaveta_6_11:=[[-887.83,-639.90,1299.67],[0.718477,0.694315,-0.039361,-0.0129874],[-1,1,-1,0],[9E+09,9E+09,9E+09,9E+09,9E+09,9E+09]];
    CONST robtarget pDepGaveta_6_21:=[[-612.28,-1051.68,1126.85],[0.71752,0.695289,-0.0138636,-0.0393256],[0,1,-1,0],[9E+09,9E+09,9E+09,9E+09,9E+09,9E+09]];
    CONST robtarget pDepGaveta_6_31:=[[-612.26,-1436.70,1078.08],[0.717526,0.695283,-0.0138581,-0.0393292],[0,1,-1,0],[9E+09,9E+09,9E+09,9E+09,9E+09,9E+09]];
    CONST robtarget pDepGaveta_6_41:=[[-612.26,-1491.41,1059.36],[0.71753,0.695278,-0.0138587,-0.0393387],[0,1,-1,0],[9E+09,9E+09,9E+09,9E+09,9E+09,9E+09]];
    CONST robtarget pDepGaveta_6_51:=[[-612.24,-1634.60,1059.35],[0.717527,0.695281,-0.0138553,-0.0393363],[0,1,-1,0],[9E+09,9E+09,9E+09,9E+09,9E+09,9E+09]];
    CONST robtarget pDepGaveta_6_61:=[[-689.98,-1634.60,1059.36],[0.71753,0.695277,-0.0138582,-0.0393362],[0,1,-1,0],[9E+09,9E+09,9E+09,9E+09,9E+09,9E+09]];
    CONST robtarget pDepGaveta_6_71:=[[-689.40,-1620.66,999.30],[0.71763,0.695227,-0.0253275,-0.0320195],[0,1,-1,0],[9E+09,9E+09,9E+09,9E+09,9E+09,9E+09]];
    CONST robtarget pDepGaveta_6_81:=[[-689.40,-1620.66,1058.84],[0.717633,0.695223,-0.0253276,-0.0320244],[0,1,-1,0],[9E+09,9E+09,9E+09,9E+09,9E+09,9E+09]];
    CONST robtarget pDepGaveta_6_91:=[[-689.43,-1220.74,1058.83],[0.717633,0.695223,-0.0253383,-0.0320325],[0,1,-1,0],[9E+09,9E+09,9E+09,9E+09,9E+09,9E+09]];
    CONST robtarget pDepGaveta_6_101:=[[-887.83,-639.91,1066.32],[0.0020033,-0.903455,-0.428667,0.00306161],[0,-1,0,0],[9E+09,9E+09,9E+09,9E+09,9E+09,9E+09]];
    CONST robtarget pRetGaveta_6_1:=[[-689.40,-1620.65,1058.82],[0.717628,0.695229,-0.0253274,-0.0320226],[0,1,-1,0],[9E+09,9E+09,9E+09,9E+09,9E+09,9E+09]];
    CONST robtarget pRetGaveta_6_11:=[[-965.55,-1348.17,1058.82],[0.717628,0.695229,-0.0253369,-0.0320263],[-1,1,-1,0],[9E+09,9E+09,9E+09,9E+09,9E+09,9E+09]];
    CONST robtarget pRetGaveta_6_21:=[[-689.41,-1620.64,945.25],[0.717631,0.695226,-0.0253295,-0.0320275],[0,1,-1,0],[9E+09,9E+09,9E+09,9E+09,9E+09,9E+09]];
    CONST robtarget pRetGaveta_6_31:=[[-689.43,-1620.63,1063.70],[0.717629,0.695227,-0.025333,-0.0320299],[0,1,-1,0],[9E+09,9E+09,9E+09,9E+09,9E+09,9E+09]];
    CONST robtarget pRetGaveta_6_41:=[[-689.45,-1546.94,1063.70],[0.717632,0.695224,-0.0253349,-0.0320324],[0,1,-1,0],[9E+09,9E+09,9E+09,9E+09,9E+09,9E+09]];
    CONST robtarget pRetGaveta_6_51:=[[-689.45,-1546.94,1107.17],[0.717633,0.695223,-0.0253351,-0.0320331],[0,1,-1,0],[9E+09,9E+09,9E+09,9E+09,9E+09,9E+09]];
    CONST robtarget pRetGaveta_6_61:=[[-689.47,-1420.87,1107.16],[0.717632,0.695224,-0.0253434,-0.0320327],[0,1,-1,0],[9E+09,9E+09,9E+09,9E+09,9E+09,9E+09]];
    CONST robtarget pRetGaveta_6_71:=[[-689.48,-1420.86,1127.23],[0.717633,0.695223,-0.0253452,-0.0320365],[0,1,-1,0],[9E+09,9E+09,9E+09,9E+09,9E+09,9E+09]];
    CONST robtarget pRetGaveta_6_81:=[[-689.48,-998.43,1127.23],[0.717631,0.695224,-0.0253476,-0.032036],[-1,1,-1,0],[9E+09,9E+09,9E+09,9E+09,9E+09,9E+09]];
    CONST robtarget pRetGaveta_6_91:=[[-1148.72,-802.12,1488.02],[0.157725,-0.703899,-0.622036,-0.304501],[0,-1,-1,0],[9E+09,9E+09,9E+09,9E+09,9E+09,9E+09]];
    CONST robtarget pRetGaveta_6_101:=[[-309.29,-759.88,1174.59],[0.243259,-0.67509,-0.655853,-0.234381],[0,-1,0,0],[9E+09,9E+09,9E+09,9E+09,9E+09,9E+09]];
    CONST robtarget MDF_p101:=[[-786.03,-814.50,1219.36],[0.114671,0.191348,0.969231,-0.104056],[-1,-2,0,1],[9E+09,9E+09,9E+09,9E+09,9E+09,9E+09]];
    CONST robtarget MDF_p111:=[[-309.29,-759.88,1174.59],[0.243259,-0.675091,-0.655854,-0.234379],[0,-1,0,0],[9E+09,9E+09,9E+09,9E+09,9E+09,9E+09]];
    CONST robtarget MDF_p121:=[[-444.14,-994.25,1198.14],[0.169061,-0.703455,-0.686189,0.0755858],[0,-1,0,0],[9E+09,9E+09,9E+09,9E+09,9E+09,9E+09]];
    CONST robtarget MDF_p131:=[[-918.44,-793.08,1198.14],[0.169067,-0.703463,-0.686181,0.0755792],[0,-1,-1,0],[9E+09,9E+09,9E+09,9E+09,9E+09,9E+09]];
    CONST robtarget MDF_p141:=[[-1167.58,-379.70,1502.84],[0.0139596,0.2323,0.879573,-0.414962],[-1,-2,-1,1],[9E+09,9E+09,9E+09,9E+09,9E+09,9E+09]];
    CONST robtarget pDepGaveta_3:=[[-693.25,-1633.70,2030.50],[0.70562,0.70809,-0.00183811,-0.0265562],[0,0,0,0],[9E+09,9E+09,9E+09,9E+09,9E+09,9E+09]];
    CONST robtarget pDepGaveta_4:=[[-1362.27,-1526.98,2038.85],[0.712891,0.700426,-0.00886317,-0.0333322],[-1,0,0,0],[9E+09,9E+09,9E+09,9E+09,9E+09,9E+09]];
    CONST robtarget pDepGaveta_4_111:=[[-1362.31,-1350.98,2140.09],[0.712887,0.70043,-0.00886857,-0.0333361],[-1,0,0,0],[9E+09,9E+09,9E+09,9E+09,9E+09,9E+09]];
    CONST robtarget pRetGaveta_4_111:=[[-1367.74,-1529.01,2088.83],[0.71763,0.695226,-0.0253439,-0.0320312],[-1,0,0,0],[9E+09,9E+09,9E+09,9E+09,9E+09,9E+09]];
    CONST robtarget pRetGaveta_3_111:=[[-693.14,-1637.83,2085.10],[0.71763,0.695229,-0.025304,-0.0320083],[0,0,0,0],[9E+09,9E+09,9E+09,9E+09,9E+09,9E+09]];
    !
    !*********************************************************
    ! Routine:  Main()
    !*********************************************************
    PROC Main()
        !
        ROB_Reset;
        ROB_Interrupt;
        ConfL\On;
        USR_Print(s_LineaVuota{nIdioma});
        ROB_Homing;
        ROB_SetForaArea;
        ROB_Setup;
        nMaxRobSpeed:=MaxRobSpeed();

        WHILE TRUE DO
            ROB_ControleAr;
            Set DO_W09_AbrirGarra;
            nTipoPcNaPinca:=0;
            bPcColocada:=TRUE;
            IF DI_P016_MdfFimCiclo=1 THEN
                ROB_FimCiclo;
            ENDIF
            ROB_SetForaArea;
            MDF_EsperaInsAutIny;
            VelSet nOverVel,nVelMax;
            mMDF_Espera;
            MDF_EsperaEntrada;
            IF bMassaloteKo=FALSE THEN
                mMDF_Pega;
                IF bInjecaoKo=FALSE THEN
                    mMDF_Saida;
                ELSE
                    mMDF_ErrSaida;
                ENDIF
            ENDIF
            IF bMassaloteKo=FALSE AND bInjecaoKo=FALSE THEN
                mSNS_ControlPc;
                IF bHbltcCicloSpec=FALSE THEN
                    DEP_GestColocStd;
                ELSE
                    DEP_GestColocNonStd;
                ENDIF
            ENDIF
            mROB_Home;
            IF bMassaloteKo=TRUE OR bInjecaoKo=TRUE THEN
                MDF_AnomaliaExtracao;
            ENDIF
            USR_Print(s_LineaVuota{nIdioma});
        ENDWHILE

    ENDPROC

    !*********************************************************
    ! Routine:  DEP_GestColocStd()
    !*********************************************************
    PROC DEP_GestColocStd()
        !Se esfriamento habilitado e peca boa e nao incompleta ou esfria rejeicao...
        IF bHbltcEsfriamento=TRUE AND ((bPcBoaDeMdf=TRUE AND bPcIncompleta=FALSE) OR bHbltcEnfriaRejeicao=TRUE) THEN
            !mENF_Cuba;
            fDepositaGaveta := TRUE;
            mDep_Gavetas;
        ENDIF
        !Verifica se existe peca no intermediario
        bErrSnsIntColoc:=FALSE;
        !SE intermediario habilitado e sensor intermediario habilitado e sensor do intermediario...
        IF (bHbltcUtilInt=TRUE AND bHbltcSnsUtilInt=TRUE AND DI_W17_SnsUtilIntermedio=1) THEN
            bErrSnsIntColoc:=TRUE;
            ROB_AlarmeAcustico(2);
            USR_Print(s_UtilOccupato{nIdioma});
            WaitTime nTempoMensAnom;
            !Ponto Intermediario
            !MoveJ HomeBoaColoc,v4000,z100,USR_toolGarra\WObj:=wobjMDF;
            !mDEP_PcBoaColoc;
            !MRet_Gavetas;
            GOTO EndProcess;
        ENDIF
        !Se estiver livre, verifica se vai continuar o processo
        IF (bPcRejeicaoDeMdf=FALSE AND bPcIncompleta=FALSE AND bErrSnsIntColoc=FALSE) THEN
            !Se for utilizar o intermediario, rotina de coloca e pega
            IF bHbltcUtilInt=TRUE THEN
                !Coloca e retira do utilitario
                !mDEP_UtilIntColoc;
                !mDEP_UtilIntPega;
                !Substituindo pelas gavetas
                !Nessa fase, o robo ir? fazer a inversao da peca
                !antes de entrar na prensa
                !Verificar aqui se sera necessario o dispositivo
                !Obrigar o robo a retirar a peca da prensa e colocar na esteira
                !apos, pegar outra peca das gavetas para prensar
                MRet_Gavetas;
                fRetiraGaveta := TRUE;
                !
            ENDIF
            !Inicia verificacoes e rotina da prensa
            IF (bHbltcPrensaColoc=TRUE AND bQualidade=FALSE AND bErrSnsIntColoc=FALSE) THEN
                USR_Print(s_CicloPrensa{nIdioma});
                IF DI_P309_05_HbltcPrensa=1 THEN
                    bPrnOkColoc:=PrensaCtrlColoc();
                    IF bPrnOkColoc=TRUE THEN
                        mDEP_PrnColoc;
                        IF (bHbltcPrensaPega=TRUE AND bPrnOkColoc=TRUE AND bPrnErrStart1=FALSE) THEN
                            bPrnOkPega:=PrensaCtrlPega();
                            IF bPrnOkPega=TRUE THEN
                                mDEP_PrnPega;
                                mDEP_PcPrensadaColoc;
                            ENDIF
                        ENDIF
                    ENDIF
                ENDIF
            ENDIF

            IF (bHbltcPrensaColoc=TRUE AND bQualidade=FALSE AND DI_P309_05_HbltcPrensa=0) THEN
                ROB_AlarmeAcustico(2);
                USR_Print(s_PrensaNaoInserido{nIdioma});
            ENDIF

            IF bPcColocada=FALSE THEN
                mDEP_PcBoaColoc;
            ENDIF

        ELSE
            mDEP_PcRejeicaoColoc;
        ENDIF
        EndProcess:
    ENDPROC

    !==============================================
    !    LISTA DE VARIAVEIS A SEREM INSERIDAS
    !==============================================

    !PERS BOOL fGavetaPronta{5}:=[FALSE,FALSE,FALSE,FALSE,FALSE];
    !PERS NUM Gaveta;
    !PERS CLK clkTempoGaveta{6}:=[0,0,0,0,0,0];
    !
    !PERS BOOL fGavetaVazia{6}:=[FALSE,FALSE,FALSE,FALSE,FALSE];

    !num nContador;
    !DI_R001_Gaveta_1
    !DI_R002_Gaveta_2
    !DI_R003_Gaveta_3
    !DI_R004_Gaveta_4
    !DI_R005_Gaveta_5
    !DI_R006_Gaveta_6

    !PERS BOOL fCtrlGavetaVazia:= FALSE;
    !PERS NUM nHistoricoGavetas{3}:=[1,2,6];

    !=====================================
    !  Reseta o tempo da peca na gaveta
    !=====================================

    PROC resetTempoPecaGaveta(num Gaveta)

        nTempoGaveta{Gaveta}:=0;
        !;clkStop clkTempoGaveta{Gaveta};
        !;clkReset clkTempoGaveta{Gaveta};
        !;clkStart clkTempoGaveta{Gaveta};

    ENDPROC

    !====================================
    !  Verifica o tempo que a peca estana gaveta
    ! E retorna se esta pronta ou nao

    PROC verificaTempoGaveta(num Gaveta)

        !clkStop TempoGaveta{Gaveta};
        !nTempoGaveta{Gaveta} := clkRead(TempoGaveta{Gaveta});
        !clkStart TempoGaveta{Gaveta};
        IF nTempoGaveta{Gaveta}>=300 THEN
            fGavetaPronta{Gaveta}:=TRUE;
        ELSE
            fGavetaPronta{Gaveta}:=FALSE;
        ENDIF

    ENDPROC

    PROC checaGavetaVazia()
        IF DI_W10_Berco_01=0 THEN
            fGavetaVazia{1}:=TRUE;
        ENDIF
        IF DI_W11_Berco_02=0 THEN
            fGavetaVazia{2}:=TRUE;
        ENDIF
        IF DI_W12_Berco_03=0 THEN
            fGavetaVazia{3}:=TRUE;
        ENDIF
        IF DI_W13_Berco_04=0 THEN
            fGavetaVazia{4}:=TRUE;
        ENDIF
        IF DI_W14_Berco_05=0 THEN
            fGavetaVazia{5}:=TRUE;
        ENDIF
        IF DI_W15_Berco_06=0 THEN
            fGavetaVazia{6}:=TRUE;
        ENDIF
    ENDPROC

    !====================================================================
    !   Rotina: mDep_Gavetas
    !   Desc.:  Rotina que gerencia todo o processo de carga das gavetas
    !====================================================================

    PROC MDep_Gavetas()

        checaGavetaVazia;

        FOR nGavetaVazia FROM 1 TO 6 DO
            IF fGavetaVazia{nGavetaVazia} AND fDepositaGaveta THEN
                !
                CallByVar "mDepGaveta_",nGavetaVazia;
                fDepositaGaveta := FALSE;
                Break;
            ENDIF
        ENDFOR

        !WHILE fCtrlGavetaVazia<>FALSE DO
            !!Loop para verificar qual gaveta esta vazia
            !!Salvar na variavel gaveta
!
!
        !ENDWHILE

    ENDPROC

        !====================================================================
    !   Rotina: mDep_Gavetas
    !   Desc.:  Rotina que gerencia todo o processo de descarga das gavetas
    !========================================================================

    PROC MRet_Gavetas()

        checaGavetaVazia;

        FOR nGavetaVazia FROM 6 TO 1 DO
            IF (fGavetaVazia{nGavetaVazia} = FALSE AND fRetiraGaveta) THEN
                !
                CallByVar "mRetiraGaveta_",nGavetaVazia;
                nRetirouDaGaveta := nGavetaVazia;
                fRetiraGaveta := FALSE;
                !
            ENDIF
        ENDFOR

        !WHILE fCtrlGavetaVazia<>FALSE DO
            !!Loop para verificar qual gaveta esta vazia
            !!Salvar na variavel gaveta
!
!
        !ENDWHILE

    ENDPROC

    !*********************************************************
    ! Routine:  DEP_GestColocNonStd()
    ! Nota:		solamente con bHbltcPrensaPega y bHbltcUtilInt
    !*********************************************************
    PROC DEP_GestColocNonStd()

        IF bHbltcEsfriamento=TRUE AND ((bPcBoaDeMdf=TRUE AND bPcIncompleta=FALSE) OR bHbltcEnfriaRejeicao=TRUE) THEN
            mENF_Cuba;
        ENDIF

        bErrSnsIntColoc:=FALSE;
        IF (bHbltcUtilInt=TRUE AND bHbltcSnsUtilInt=TRUE AND DI_W17_SnsUtilIntermedio=1) THEN
            bErrSnsIntColoc:=TRUE;
            ROB_AlarmeAcustico(2);
            USR_Print(s_UtilOccupato{nIdioma});
            WaitTime nTempoMensAnom;
            !Ponto Intermediario
            MoveJ HomeBoaColoc,v4000,z100,USR_toolGarra\WObj:=wobjMDF;
            mDEP_PcBoaColoc;
            GOTO EndProcess;
        ENDIF

        IF (bPcRejeicaoDeMdf=FALSE AND bPcIncompleta=FALSE AND bErrSnsIntColoc=FALSE) THEN

            mDEP_UtilIntColoc;

            IF (bHbltcPrensaPega=TRUE AND DI_P309_05_HbltcPrensa=1) THEN
                USR_Print(s_CicloPrensa{nIdioma});
                bPrnOkPega:=PrensaCtrlPega();
                IF bPrnOkPega=TRUE THEN
                    mDEP_PrnPega;
                    mDEP_PcPrensadaColoc;
                ENDIF
            ENDIF

            mDEP_UtilIntPega;

            IF (bHbltcPrensaColoc=TRUE AND bQualidade=FALSE) THEN
                USR_Print(s_CicloPrensa{nIdioma});
                IF DI_P309_05_HbltcPrensa=1 THEN
                    bPrnOkColoc:=PrensaCtrlColoc();
                    IF bPrnOkColoc=TRUE THEN
                        mDEP_PrnColoc;
                    ENDIF
                ENDIF
            ENDIF

            IF (bHbltcPrensaColoc=TRUE AND bQualidade=FALSE AND DI_P309_05_HbltcPrensa=0) THEN
                ROB_AlarmeAcustico(2);
                USR_Print(s_PrensaNaoInserido{nIdioma});
            ENDIF

            IF bPcColocada=FALSE THEN
                mDEP_PcBoaColoc;
            ENDIF

        ELSE
            mDEP_PcRejeicaoColoc;
        ENDIF
        EndProcess:
    ENDPROC

    !*********************************************************
    ! Routine:  ROB_Interrupt()
    !*********************************************************
    PROC ROB_Interrupt()

        IDelete intVel0;
        IDelete intVelStd;
        IDelete intMslKo;

        IDelete intQualidade;
        CONNECT intQualidade WITH TR_Qualidade;
        ISignalDI DI_V02_ReqQualidade,1,intQualidade;

    ENDPROC

    TRAP TR_Qualidade
        bQualidade:=TRUE;
        Set DO_W02_LuzAmarelo;
        ROB_AlarmeAcustico(2);
        USR_Print(s_ReqQualita{nIdioma});
    ENDTRAP

    !*********************************************************
    ! Routine:  ROB_HomingInterrupt()
    !*********************************************************
    PROC ROB_HomingInterrupt()

        IDelete intVel0;
        CONNECT intVel0 WITH TR_Vel0;
        ISignalDI DI_P305_01_StartCiclo,0,intVel0;

        IDelete intVelStd;
        CONNECT intVelStd WITH TR_VelStd;
        ISignalDI DI_P305_01_StartCiclo,1,intVelStd;

        SpeedRefresh 100;

    ENDPROC

    TRAP TR_Vel0
        SpeedRefresh 0;
        IF (bPegaCtrlMdf=TRUE AND DI_P006_MoldeAberto=0) THEN
            USR_Print(s_MancaStampoAperto{nIdioma});
        ENDIF
    ENDTRAP

    TRAP TR_VelStd
        SpeedRefresh 100;
    ENDTRAP

    !*********************************************************
    ! Routine:  ROB_Reset()
    !*********************************************************
    PROC ROB_Reset()

        Reset DO_P003_StartPulver;
        Reset DO_P006_AnomaliaRobo;
        Reset DO_P007_StartExpulsAdel;
        Reset DO_P008_StartExpulsAtras;
        Reset DO_P010_PrgCarregado;
        Reset DO_P011_PrgExistente;
        Reset DO_P012_PrgAusente;
        Reset DO_P013_OkFecharMdf;
        Reset DO_P014_PulverRadPM;
        Reset DO_P015_PcIncompleta;
        Reset DO_P017_PrgGuardado;
        Reset DO_P018_PulverEmbolo;
        Reset DO_P019_PulverRadPF;
        Reset DO_P021_ErrSnsStartPulver;
        Reset DO_P022_FimCiclo;
        Reset DO_P064_FimCicloInsertos;
        Reset DO_P242_PrnStartAposColoc;
        Reset DO_P243_PrnStartAposPega;
        Reset DO_W02_LuzAmarelo;
        Reset DO_W03_AlarmeAcustico;
        Reset DO_W08_StartEsteiraBoa;
        Reset DO_V05_MdfForaAreaTrab_User;
        Reset DO_V06_PrensaForaAreaTrab_User;
        Reset DO_V08_LuzVermelha;

        bQualidade:=FALSE;
        bPcIncompleta:=FALSE;
        bPcRejeicaoDeMdf:=FALSE;
        bPcBoaDeMdf:=FALSE;
        bInjecaoKo:=FALSE;
        bPcColocada:=TRUE;
        bPrnOkColoc:=FALSE;
        bPrnOkPega:=FALSE;
        bPegaCtrlMdf:=FALSE;

        ClkReset timerEXT;
        ClkReset timerROB;
        ClkReset timerMDF;

        nTipoPcNaPinca:=0;

        FOR i FROM 1 TO 11 DO
            stVideo{i}:=" ";
        ENDFOR

    ENDPROC

    !*********************************************************
    ! Routine:  ROB_Homing()
    !*********************************************************
    PROC ROB_Homing()

        VAR bool bRobEmHome;
        VAR bool bRobEnEspera;

        ROB_HomingInterrupt;

        aaa:
        USR_toolRestore:=CTool();
        ROB_pStartHoming:=CRobT(\Tool:=USR_toolRestore\WObj:=wobjMDF);
        ROB_jStartHoming:=CJointT();

        bRobEmHome:=CtrlRobPos(ROB_pHome);
        bRobEnEspera:=CtrlRobPos(MDF_pEspera);

        IF (bRobEmHome=FALSE) AND (bRobEnEspera=FALSE) THEN
            USR_Print(s_LineaVuota{nIdioma});
            USR_Print(s_PremiStart1{nIdioma});
            USR_Print(s_PremiStart2{nIdioma});
        ENDIF

        WaitTime\inpos,0;
        SoftDeact;
        ROB_GarraFechar;
        ROB_GarraAbrir;
        nTipoPcNaPinca:=0;
        bPcColocada:=TRUE;

        IF bRobEmHome OR bRobEnEspera THEN
            ROB_nPosRobo:=0;
        ELSEIF ROB_jStartHoming.robax.rax_1>=(njMdfMin) AND ROB_jStartHoming.robax.rax_1<(njMdfMax) THEN
            ROB_nPosRobo:=1;
            USR_Print(s_RiprPfo{nIdioma});
        ELSEIF ROB_jStartHoming.robax.rax_1>=(njUtilMin) AND ROB_jStartHoming.robax.rax_1<(njUtilMax) THEN
            ROB_nPosRobo:=2;
            USR_Print(s_RiprUtil{nIdioma});
        ELSEIF ROB_jStartHoming.robax.rax_1>=(njCubaMin) AND ROB_jStartHoming.robax.rax_1<(njCubaMax) THEN
            ROB_nPosRobo:=3;
            USR_Print(s_RiprRaffr{nIdioma});
        ELSEIF ROB_jStartHoming.robax.rax_1>=(njRampaMin) AND ROB_jStartHoming.robax.rax_1<(njRampaMax) THEN
            ROB_nPosRobo:=4;
            USR_Print(s_RiprBuoni{nIdioma});
        ELSEIF ROB_jStartHoming.robax.rax_1>=(njPrensaMin) AND ROB_jStartHoming.robax.rax_1<(njPrensaMax) THEN
            ROB_nPosRobo:=5;
            USR_Print(s_RiprPrensa{nIdioma});
        ELSE
            USR_Print(s_RiprErrore{nIdioma});
            WaitTime 3;
            ROB_nPosRobo:=99;
        ENDIF

        TEST ROB_nPosRobo
        CASE 0:
            ! HOME POSITION // ESPERA ENTRADA
            IDelete intVel0;
            IDelete intVelStd;
            SpeedRefresh 25;
            MoveL ROB_pHome,v1000,fine,USR_toolRestore\wobj:=wobjMDF;
            SpeedRefresh 100;
        CASE 1:
            ! MDF (M?quina De FundiCAO inyectada)
            IF ROB_jStartHoming.robax.rax_2>0 THEN
                MoveL RelTool(ROB_pStartHoming,0,40,0),v100,z1,USR_toolRestore\wobj:=wobjMDF;
                MoveL MDF_p02,v100,z1,USR_toolRestore\wobj:=wobjMDF;
                MoveJ MDF_p01,v100,z1,USR_toolGarra\WObj:=wobjMDF;
            ENDIF
            MoveJ MDF_pEspera,v100,z1,USR_toolRestore\wobj:=wobjMDF;
            MoveL ROB_pHome,v100,fine,USR_toolRestore\wobj:=wobjMDF;
            WaitDI DI_P305_01_StartCiclo,0;
            WaitDI DI_P305_01_StartCiclo,1;
        CASE 2:
            ! UTIL
            MoveJ UTL_p62,v100,z1,USR_toolGarra\WObj:=wobjMDF;
            MoveJ ROB_pHome,v100,fine,USR_toolRestore\wobj:=wobjMDF;
            WaitDI DI_P305_01_StartCiclo,0;
            WaitDI DI_P305_01_StartCiclo,1;
        CASE 3:
            ! CUBA DE AGUA
            MoveJ Offs(ROB_pStartHoming,0,0,300),v100,z1,USR_toolRestore\wobj:=wobjMDF;
            MoveJ ENF_p23,v100,z1,USR_toolGarra\WObj:=wobjMDF;
            MoveJ ROB_pHome,v100,fine,USR_toolRestore\wobj:=wobjMDF;
            WaitDI DI_P305_01_StartCiclo,0;
            WaitDI DI_P305_01_StartCiclo,1;
        CASE 4:
            ! RAMPA BUENA/CALIDAD
            MoveJ Offs(ROB_pStartHoming,0,0,300),v100,z1,USR_toolRestore\wobj:=wobjMDF;
            MoveJ BUE_p14,v100,z1,USR_toolGarra\WObj:=wobjMDF;
            MoveJ ROB_pHome,v100,fine,USR_toolRestore\wobj:=wobjMDF;
            WaitDI DI_P305_01_StartCiclo,0;
            WaitDI DI_P305_01_StartCiclo,1;
        CASE 5:
            ! PRENSA
            MoveJ Offs(ROB_pStartHoming,0,0,50),v100,z1,USR_toolRestore\wobj:=wobjMDF;
            MoveJ PRN_p14,v100,z1,USR_toolGarra\WObj:=wobjMDF;
            MoveJ ROB_pHome,v100,fine,USR_toolRestore\wobj:=wobjMDF;
            WaitDI DI_P305_01_StartCiclo,0;
            WaitDI DI_P305_01_StartCiclo,1;
        CASE 99:
            ! POSICAO DESCONOCIDA: MOVIMIENTO MANUAL!
            Stop;
            GOTO aaa;
        DEFAULT:
            IDelete intVel0;
            IDelete intVelStd;
            SpeedRefresh 100;
            EXIT;
        ENDTEST

        IDelete intVel0;
        IDelete intVelStd;
        SpeedRefresh 100;

    ENDPROC

    !*********************************************************
    ! Routine:  ROB_SetForaArea()
    !*********************************************************
    PROC ROB_SetForaArea()

        Set DO_V05_MdfForaAreaTrab_User;
        Set DO_V06_PrensaForaAreaTrab_User;

    ENDPROC

    !*********************************************************
    ! Routine:  ROB_GarraAbrir
    !*********************************************************
    PROC ROB_GarraAbrir()

        WaitTime\inpos,0;
        Set DO_W09_AbrirGarra;
        WaitTime nTempoGarraAbrir;
        GripLoad load0;

    ENDPROC

    !*********************************************************
    ! Routine:  ROB_GarraFechar
    !*********************************************************
    PROC ROB_GarraFechar()

        WaitTime\inpos,0;
        Reset DO_W09_AbrirGarra;
        WaitTime nTempoGarraFechar;
        GripLoad loadPeca;

    ENDPROC

    !*********************************************************
    ! Routine:  ROB_AlarmeAcustico()
    ! Input parameter:  ancho de pulso
    !*********************************************************
    PROC ROB_AlarmeAcustico(
			num nLength)

        Reset DO_W03_AlarmeAcustico;
        PulseDO\PLength:=nLength,DO_W03_AlarmeAcustico;

    ENDPROC

    !*********************************************************
    ! Routine:  ROB_ControleAr()
    !*********************************************************
    PROC ROB_ControleAr()
        VAR bool bArKo:=TRUE;

        WHILE bArKo=TRUE DO
            WaitDI DI_W21_PresAr,1\MaxTime:=nTempoMaxDIAr\TimeFlag:=bArKo;
            IF bArKo=TRUE THEN
                Set DO_V08_LuzVermelha;
                ROB_AlarmeAcustico(2);
                Reset DO_P042_ErrPresAr;
                PulseDO\PLength:=1,DO_P042_ErrPresAr;
                USR_Print(s_PressioneAria{nIdioma});
                USR_Print(s_AttesaReset{nIdioma});
                WaitDI DI_V01_ResetAllRob,1;
            ENDIF
            Reset DO_V08_LuzVermelha;
        ENDWHILE

    ENDPROC

    !*********************************************************
    ! Routine:  ROB_FimCiclo()
    !*********************************************************
    PROC ROB_FimCiclo()
        VAR bool bTemp:=FALSE;

        IF (bHbltcCicloSpec=TRUE AND bHbltcPrensaPega=TRUE AND DI_P309_05_HbltcPrensa=1) THEN
            USR_Print(s_CicloPrensa{nIdioma});
            bPrnOkPega:=PrensaCtrlPega();
            IF bPrnOkPega=TRUE THEN
                mDEP_PrnPega;
                mDEP_PcPrensadaColoc;
                mROB_Home;
            ENDIF
        ENDIF

        WaitTime\inpos,0;

        ! espera fine de ciclo de prensa (si activada)
        IF (bHbltcPrensaColoc=TRUE AND DI_P309_05_HbltcPrensa=1 AND DI_P240_PrnAuto=1) THEN
            USR_MsgWaitDI DI_P242_PrnOkColoc,s_AttesaFineCicloPrensa{nIdioma};
            WaitUntil(DI_P242_PrnOkColoc=1 OR DI_P243_PrnOkPega=1)\MaxTime:=nTempoMaxDIPrnFimCiclo\TimeFlag:=bTemp;
        ENDIF

        USR_Print(s_OkAperturaPorta{nIdioma});
        Reset DO_P022_FimCiclo;
        PulseDO\PLength:=2,DO_P022_FimCiclo;
        WaitTime 1;
        ! Reset DO_V00_MotorOff;
        ! PulseDO\PLength:=0.2,DO_V00_MotorOff;
        WaitTime 1;

    ENDPROC

    !*********************************************************
    ! Routine:  mROB_Home()
    !*********************************************************
    PROC mROB_Home()

        USR_Print(s_RoboHome{nIdioma});
        !MoveL ROB_pHome, vmax, z5, USR_toolGarra\wobj:=wobjMDF;
        MoveJ ROB_pHome,vmax,z5,USR_toolGarra\WObj:=wobjMDF;
        !MoveJ [[-310.41,-957.32,1307.40],[0.0503054,-0.713482,-0.697746,-0.0395422],[0,-1,0,0],[9E+09,9E+09,9E+09,9E+09,9E+09,9E+09]], vmax, z5, USR_toolGarra\WObj:=wobjMDF;

    ENDPROC

    !*********************************************************
    ! Routine:  mMDF_Espera()
    !*********************************************************
    PROC mMDF_Espera()

        USR_Print(s_RoboDavantiPfo{nIdioma});
        MoveJ MDF_pEsperaprevio,vmax,z5,USR_toolGarra\WObj:=wobjMDF;
        MoveJ MDF_pEspera,vmax,z5,USR_toolGarra\WObj:=wobjMDF;

    ENDPROC

    !*********************************************************
    ! Routine:  MDF_EsperaInsAutIny()
    !*********************************************************
    PROC MDF_EsperaInsAutIny()

        ClkStop timerROB;
        ROB_nTimerROB:=ClkRead(timerROB);

        WHILE DI_P000_RoboAtivado=0 OR DI_P001_MdfCicloAuto=0 OR DI_P002_InjecaoOk=0 DO
            IF DI_P000_RoboAtivado=0 THEN
                USR_MsgWaitDI DI_P000_RoboAtivado,s_RoboInserito{nIdioma};
                WaitDI DI_P000_RoboAtivado,1;
            ELSEIF DI_P001_MdfCicloAuto=0 THEN
                USR_MsgWaitDI DI_P001_MdfCicloAuto,s_AutomaticoPfo{nIdioma};
                WaitDI DI_P001_MdfCicloAuto,1;
            ELSEIF DI_P002_InjecaoOk=0 THEN
                USR_MsgWaitDI DI_P002_InjecaoOk,s_AttesaPrelievoPfo{nIdioma};
                WaitDI DI_P002_InjecaoOk,1;
            ENDIF
        ENDWHILE

    ENDPROC

    !*********************************************************
    ! Routine:  MDF_EsperaEntrada()
    !*********************************************************
    PROC MDF_EsperaEntrada()

        bMassaloteKo:=FALSE;
        IDelete intMslKo;
        CONNECT intMslKo WITH TR_MtzNonOk;
        ISignalDI DI_P013_MassaloteNonOk,1,intMslKo;

        WHILE (DI_P000_RoboAtivado=0 OR DI_P001_MdfCicloAuto=0 OR DI_P006_MoldeAberto=0 OR DI_P002_InjecaoOk=0 OR DI_P005_ExpulsAtras=0 OR DI_P009_PortaAberta=0) AND bMassaloteKo=FALSE DO
            IF DI_P000_RoboAtivado=0 THEN
                USR_MsgWaitDI DI_P000_RoboAtivado,s_RoboInserito{nIdioma};
                WaitDI DI_P000_RoboAtivado,1;
            ELSEIF DI_P001_MdfCicloAuto=0 THEN
                USR_MsgWaitDI DI_P001_MdfCicloAuto,s_AutomaticoPfo{nIdioma};
                WaitDI DI_P001_MdfCicloAuto,1;
            ELSEIF DI_P002_InjecaoOk=0 THEN
                USR_MsgWaitDI DI_P002_InjecaoOk,s_AttesaPrelievoPfo{nIdioma};
                WaitDI DI_P002_InjecaoOk,1;
            ELSEIF DI_P005_ExpulsAtras=0 THEN
                USR_MsgWaitDI DI_P005_ExpulsAtras,s_AttesaEstrazInd{nIdioma};
                WaitDI DI_P005_ExpulsAtras,1;
            ELSEIF DI_P009_PortaAberta=0 THEN
                USR_MsgWaitDI DI_P009_PortaAberta,s_AttesaCancAperto{nIdioma};
                WaitDI DI_P009_PortaAberta,1;
            ELSEIF DI_P006_MoldeAberto=0 THEN
                USR_MsgWaitDI DI_P006_MoldeAberto,s_AttesaAperturaPfo{nIdioma};
                WaitDI DI_P006_MoldeAberto,1;
            ENDIF
        ENDWHILE

        IDelete intMslKo;

        ClkStop timerMDF;
        ROB_ntimerMDF:=ClkRead(timerMDF);
        ClkReset timerMDF;
        ClkStart timerMDF;
        ClkStart timerEXT;

    ENDPROC

    TRAP TR_MtzNonOk
        bMassaloteKo:=TRUE;
    ENDTRAP

    !*********************************************************
    ! Routine:  ROB_MoldeAbertoInt()
    !*********************************************************
    PROC ROB_MoldeAbertoInt()

        IDelete intVel0;
        CONNECT intVel0 WITH TR_Vel0;
        ISignalDI DI_P006_MoldeAberto,0,intVel0;

        IDelete intVelStd;
        CONNECT intVelStd WITH TR_VelStd;
        ISignalDI DI_P006_MoldeAberto,1,intVelStd;

    ENDPROC

    !*********************************************************
    ! Routine:  mMDF_Pega() Pega = Pegar
    !*********************************************************
    PROC mMDF_Pega()

        MoveL MDF_pEspera,vmax,z5,USR_toolGarra\wobj:=wobjMDF;

        bPegaCtrlMdf:=FALSE;
        IF bHbltcCtrlMoldeAberto=TRUE THEN
            ROB_MoldeAbertoInt;
            bPegaCtrlMdf:=TRUE;
        ENDIF

        bAnomSnsPulver:=FALSE;
        IF DI_W16_SnsStartPulver=1 THEN
            bAnomSnsPulver:=TRUE;
            USR_Print(s_AnomaliaSnsStartLub{nIdioma});
            ROB_AlarmeAcustico(2);
        ENDIF

        USR_Print(s_PrelievoPfo{nIdioma});
        Set DO_W09_AbrirGarra;
        nTipoPcNaPinca:=0;
        bPcColocada:=TRUE;
        Reset DO_P003_StartPulver;
        Reset DO_P013_OkFecharMdf;
        Reset DO_V05_MdfForaAreaTrab_User;

        MoveJ MDF_p01,v4000,z50,USR_toolGarra\WObj:=wobjMDF;
        MoveJ MDF_p03,v4000,z50,USR_toolGarra\WObj:=wobjMDF;

        IF bHbltcSoftservo=FALSE THEN
            Set DO_P007_StartExpulsAdel;
        ENDIF

        ConfL\Off;
        SingArea\Wrist;

        MoveL MDF_p03,v150,z50,USR_toolGarra\WObj:=wobjMDF;

        ! ===>>> POSICAO DE RETIRADA <<<===
        MoveL MDF_pPega,v300,fine,USR_toolGarra\WObj:=wobjMDF;
        ! ==================================

        ! memorizaCAO PECA buena/calidad/rechazo
        bPcRejeicaoDeMdf:=FALSE;
        bPcBoaDeMdf:=FALSE;
        IF (DI_P018_MdfStartUp=0 AND DI_P019_PcRejeicao=0 AND DI_P011_PcBoa=1 AND bQualidade=FALSE) THEN
            bPcBoaDeMdf:=TRUE;
            nTipoPcNaPinca:=1;
            USR_Print(s_GarraBuono{nIdioma});
        ELSEIF (DI_P018_MdfStartUp=0 AND DI_P019_PcRejeicao=0 AND DI_P011_PcBoa=1 AND bQualidade=TRUE) THEN
            bPcBoaDeMdf:=TRUE;
            nTipoPcNaPinca:=4;
            USR_Print(s_GarraQualita{nIdioma});
        ELSE
            bPcRejeicaoDeMdf:=TRUE;
            !Rejeicao:=Rejeicao;
            nTipoPcNaPinca:=3;
            USR_Print(s_GarraScarto{nIdioma});
        ENDIF

        USR_Print(s_EstrazionePfo{nIdioma});
        IF bHbltcSoftservo=TRUE THEN
            ! pega CON ACOMPA?AMIENTO (SOFTSERVO)
            Reset DO_W09_AbrirGarra;
            bPcColocada:=FALSE;
            ! opzione???
            ! MotionSup \Off;
            SoftAct 1,98;
            SoftAct 2,10;
            SoftAct 3,10;
            SoftAct 4,30;
            SoftAct 5,20;
            SoftAct 6,20;
            WaitTime nTempoGarraFechar;
            !Tempo espera pasaje hacia ejes soft
            Set DO_P007_StartExpulsAdel;
            USR_MsgWaitDI DI_P004_ExpulsAdel,s_EstrazioneAvanti{nIdioma};
            !MoveL [[2692.31,-365.59,1196.61],[0.998402,0.00144403,0.0559844,0.00758486],[1,-1,0,1],[9E+09,9E+09,9E+09,9E+09,9E+09,9E+09]], v300, fine, USR_toolGarra\WObj:=wobjMDF;
            WaitDI DI_P004_ExpulsAdel,1\MaxTime:=nTempoMaxDIEyecAdel\TimeFlag:=bInjecaoKo;
            SoftDeact;
            !MoveL MDF_p03, v150, fine, USR_toolGarra\WObj:=wobjMDF;
            MoveL MDF_p43,v150,fine,USR_toolGarra\WObj:=wobjMDF;
        ELSE
            ! pega SIN acompa?amiento
            WaitTime\inpos,0;
            USR_MsgWaitDI DI_P004_ExpulsAdel,s_EstrazioneAvanti{nIdioma};
            WaitDI DI_P004_ExpulsAdel,1\MaxTime:=nTempoMaxDIEyecAdel\TimeFlag:=bInjecaoKo;
            IF bInjecaoKo=FALSE THEN
                ROB_GarraFechar;
                bPcColocada:=FALSE;
            ENDIF
        ENDIF

        IF bInjecaoKo=TRUE THEN
            USR_Print(s_EstrazioneFallita{nIdioma});
            ROB_AlarmeAcustico(2);
            Set DO_V08_LuzVermelha;
            SpeedRefresh 20;
            ROB_GarraAbrir;
            nTipoPcNaPinca:=0;
            bPcColocada:=TRUE;
        ENDIF

        IF bInjecaoKo=FALSE THEN
            MDF_pTemp:=CRobT(\Tool:=USR_toolGarra\WObj:=wobjMDF);
            MoveL MDF_p03,v300,fine,USR_toolGarra\WObj:=wobjMDF;
        ENDIF
        SoftDeact;

        MoveL MDF_p03,v1000,fine,USR_toolGarra\WObj:=wobjMDF;

        SingArea\Off;
        ConfL\On;
        WaitTime\inpos,0;
        Reset DO_P007_StartExpulsAdel;

        IF bInjecaoKo=FALSE THEN
            GripLoad loadPeca;
        ENDIF
        ! opzione???
        ! MotionSup \On;

    ENDPROC

    !*********************************************************
    ! Routine:  mMDF_Saida()
    !*********************************************************
    PROC mMDF_Saida()

        USR_Print(s_UscitaPfo{nIdioma});

        MoveL\Conc,MDF_p03,v4000,z50,USR_toolGarra\WObj:=wobjMDF;
        MoveL\Conc, MDF_p11, v4000, z50, USR_toolGarra\WObj:=wobjMDF;
        MoveJ MDF_p81,v4000,z100,USR_toolGarra\WObj:=wobjMDF;
        MoveJ MDF_p91,v4000,z50,USR_toolGarra\WObj:=wobjMDF;
        !MoveJ MDF_p40,v4000,fine,USR_toolGarra\WObj:=wobjMDF;
        !MoveJ [[966.83,-187.39,1287.16],[0.573195,-0.113432,0.811301,-0.0192816],[1,-1,0,0],[9E+09,9E+09,9E+09,9E+09,9E+09,9E+09]],vmax,z100,USR_toolGarra\WObj:=wobjMDF;
        !MoveJ MDF_p12,vmax,z50,USR_toolGarra\wobj:=wobjMDF;

        bErrSnsPulver:=FALSE;
        IF bHbltcSnsAntPulver=TRUE AND bInjecaoKo=FALSE THEN
            MoveJ MDF_p30,vmax,z50,USR_toolGarra\WObj:=wobjMDF;

            USR_Print(s_ControlloFtc{nIdioma});

            ! ===>>> POSICAO de CONTROL START PULVER. <<<===
            !MoveL MDF_pControl, v3000, z10, USR_toolGarra\WObj:=wobjMDF;
            MoveJ MDF_pControl,v3000,z20,USR_toolGarra\WObj:=wobjMDF;
            ! ===============================================

            WaitTime\inpos,0.3;
            IF (DI_W16_SnsStartPulver=1 AND bAnomSnsPulver=FALSE) THEN
                Reset DO_P003_StartPulver;
                PulseDO\PLength:=1,DO_P003_StartPulver;
                ClkStop timerEXT;
                ROB_nTimerEXT:=ClkRead(timerEXT);
                ClkReset timerEXT;
                USR_Print(s_OkSnsStartLub{nIdioma});
            ELSE
                bErrSnsPulver:=TRUE;
                ROB_AlarmeAcustico(2);
                USR_Print(s_AllarmeSnsStartLub{nIdioma});
            ENDIF

            !MoveJ MDF_p30, v1000, z50, USR_toolGarra\WObj:=wobjMDF;
            MoveJ MDF_p31,vmax,z50,USR_toolGarra\WObj:=wobjMDF;
        ENDIF

        MoveJ MDF_p30,vmax,z50,USR_toolGarra\WObj:=wobjMDF;

        ! ===>>> POSICAO FUERA de la PUERTA de la M?QUINA!!! <<<===
        MoveJDO MDF_p31,vmax,z50,USR_toolGarra\WObj:=wobjMDF,DO_V05_MdfForaAreaTrab_User,1;
        !MoveJ MDF_p31, vmax, z50, USR_toolGarra\WObj:=wobjMDF;
        ! ==========================================================
        !MoveJ MDF_p101, vmax, z50, USR_toolGarra\WObj:=wobjMDF;
        !MoveJ MDF_p141, vmax, z50, USR_toolGarra\WObj:=wobjMDF;
        !MoveJ MDF_p131, vmax, z50, USR_toolGarra\WObj:=wobjMDF;
        !MoveJ MDF_p121, vmax, z50, USR_toolGarra\WObj:=wobjMDF;
        !MoveJ MDF_p111, vmax, z50, USR_toolGarra\WObj:=wobjMDF;

        IDelete intVel0;
        IDelete intVelStd;
        bPegaCtrlMdf:=FALSE;

        IF bPcRejeicaoDeMdf=TRUE THEN
            ROB_AlarmeAcustico(1);
            USR_Print(s_ScartoDcm{nIdioma});
        ENDIF

    ENDPROC

    !*********************************************************
    ! Routine:  mMDF_ErrSaida()
    !*********************************************************
    PROC mMDF_ErrSaida()

        USR_Print(s_UscitaPfo{nIdioma});

        ConfL\Off;
        SingArea\Wrist;
        ROB_GarraAbrir;
        MoveL MDF_p02,vmax,z50,USR_toolGarra\WObj:=wobjMDF;
        SingArea\Off;
        ConfL\On;
        MoveL MDF_p10,vmax,z50,USR_toolGarra\WObj:=wobjMDF;
        MoveL MDF_p11,vmax,z5,USR_toolGarra\WObj:=wobjMDF;
        MoveJ MDF_p40,vmax,z5,USR_toolGarra\WObj:=wobjMDF;
        MoveJ MDF_p12,vmax,z5,USR_toolGarra\WObj:=wobjMDF;
        MoveJ MDF_p30,vmax,z5,USR_toolGarra\WObj:=wobjMDF;
        MoveJ MDF_p31,vmax,z5,USR_toolGarra\WObj:=wobjMDF;
        MoveJ [[-94.08,-478.58,2065.27],[0.849876,0.0295538,0.0520096,-0.523577],[0,-1,0,1],[9E+09,9E+09,9E+09,9E+09,9E+09,9E+09]],vmax,z5,USR_toolGarra\WObj:=wobjMDF;
        !MoveL ROB_pHome, vmax, z5, USR_toolGarra\wobj:=wobjMDF;
        MoveJ ROB_pHome,vmax,z5,USR_toolGarra\WObj:=wobjMDF;

        WaitTime\inpos,0.5;
        Set DO_V05_MdfForaAreaTrab_User;

        IDelete intVel0;
        IDelete intVelStd;

    ENDPROC

    !*********************************************************
    ! Routine:  mSNS_ControlPc()
    !*********************************************************
    PROC mSNS_ControlPc()

        SNS_CtrlFuncionamiento;

        MoveL\Conc, SNS_p01, vmax, z100, USR_toolGarra\WObj:=wobjMDF;
        MoveJ [[-498.07,-1238.79,1630.02],[0.680913,0.0157814,0.727053,-0.0866155],[-1,-2,0,1],[9E+09,9E+09,9E+09,9E+09,9E+09,9E+09]],vmax,z100,USR_toolGarra\WObj:=wobjMDF;
        MoveJ SNS_p02,vmax,z50,USR_toolGarra\WObj:=wobjMDF;

        USR_Print(s_ControlloFtc{nIdioma});

        bErrCtrl1:=FALSE;
        bErrCtrl2:=FALSE;
        bErrCtrl3:=FALSE;
        bErrCtrl4:=FALSE;
        bPcIncompleta:=FALSE;

        ! ===>>> 1a POSICAO de CONTROL SENSORES <<<===
        MoveL SNS_pControl1,v500,fine,USR_toolGarra\WObj:=wobjMDF;
        ! =============================================
        WaitTime\inpos,0.3;
        SNS_CtrlPeca;
        bErrCtrl1:=bErrCtrlSns;

        !IF bErrCtrlSns=FALSE THEN
        !	! ===>>> 2a POSICAO de CONTROL SENSORES <<<===
        !	MoveL SNS_pControl2, v500, fine, USR_toolGarra\WObj:=wobjMDF;
        !	! =============================================
        !	WaitTime\InPos, 0.3;
        !	SNS_CtrlPeca;
        !	bErrCtrl2:=bErrCtrlSns;
        !ENDIF

        !IF bErrCtrlSns=FALSE THEN
        !	! ===>>> 3a POSICAO de CONTROL SENSORES <<<===
        !	MoveL SNS_pControl3, v500, fine, USR_toolGarra\WObj:=wobjMDF;
        !	! =============================================
        !	WaitTime\InPos, 0.3;
        !	SNS_CtrlPeca;
        !	bErrCtrl3:=bErrCtrlSns;
        !ENDIF

        !IF bErrCtrlSns=FALSE THEN
        !	! ===>>> 4a POSICAO de CONTROL SENSORES <<<===
        !	MoveL SNS_pControl4, v500, fine, USR_toolGarra\WObj:=wobjMDF;
        !	! =============================================
        !	WaitTime\InPos, 0.3;
        !	SNS_CtrlPeca;
        !	bErrCtrl4:=bErrCtrlSns;
        !ENDIF

        ! resultado final de todos los controles
        bPcIncompleta:=bErrCtrl1 OR bErrCtrl2 OR bErrCtrl3 OR bErrCtrl4;

        ! start pulverizador
        IF bPcIncompleta=FALSE THEN
            Reset DO_P003_StartPulver;
            PulseDO\PLength:=1,DO_P003_StartPulver;
        ENDIF

        ! cron?metro tempo extra??o
        IF (bHbltcSnsAntPulver=FALSE OR bErrSnsPulver=TRUE) THEN
            ClkStop timerEXT;
            ROB_nTimerEXT:=ClkRead(timerEXT);
            ClkReset timerEXT;
        ENDIF

        ! anomal?a de control funcionamiento sensores
        IF bSnsDefect=TRUE THEN
            bPcIncompleta:=TRUE;
        ENDIF

        ! opCAO: non rechazo PECAs incompletas
        IF bHbltcGuardarIncompl=TRUE THEN
            bPcIncompleta:=FALSE;
        ENDIF

        ! anomal?a de sensor start anticipado pulverizador
        IF (bErrSnsPulver=TRUE OR bAnomSnsPulver=TRUE) THEN
            Reset DO_P021_ErrSnsStartPulver;
            PulseDO\PLength:=1,DO_P021_ErrSnsStartPulver;
        ENDIF

        MDF_Start;
        MoveJ SNS_p02,vmax,z50,USR_toolGarra\WObj:=wobjMDF;

        MoveJ SNS_p10,vmax,z50,USR_toolGarra\WObj:=wobjMDF;
        MoveJ SNS_p20,vmax,z50,USR_toolGarra\WObj:=wobjMDF;
        MoveJ SNS_p11,vmax,z100,USR_toolGarra\WObj:=wobjMDF;

    ENDPROC

    !*********************************************************
    ! Routine:  SNS_CtrlFuncionamiento()
    !*********************************************************
    PROC SNS_CtrlFuncionamiento()
        VAR errnum errvar;
        VAR num nKey:=0;

        USR_Print(s_FunzionalitaFtc{nIdioma});
        check:
        bSnsDefect:=FALSE;
        FOR i FROM 1 TO 10 DO
            nSnsDefect{i}:=0;
        ENDFOR

        IF bHbltcSns01=TRUE AND DI_W00_Sns01=1 THEN
            bSnsDefect:=TRUE;
            nSnsDefect{1}:=1;
        ENDIF
        IF bHbltcSns02=TRUE AND DI_W01_Sns02=1 THEN
            bSnsDefect:=TRUE;
            nSnsDefect{2}:=1;
        ENDIF
        IF bHbltcSns03=TRUE AND DI_W02_Sns03=1 THEN
            bSnsDefect:=TRUE;
            nSnsDefect{3}:=1;
        ENDIF
        IF bHbltcSns04=TRUE AND DI_W03_Sns04=1 THEN
            bSnsDefect:=TRUE;
            nSnsDefect{4}:=1;
        ENDIF
        IF bHbltcSns05=TRUE AND DI_W04_Sns05=1 THEN
            bSnsDefect:=TRUE;
            nSnsDefect{5}:=1;
        ENDIF
        IF bHbltcSns06=TRUE AND DI_W05_Sns06=1 THEN
            bSnsDefect:=TRUE;
            nSnsDefect{6}:=1;
        ENDIF
        IF bHbltcSns07=TRUE AND DI_W06_Sns07=1 THEN
            bSnsDefect:=TRUE;
            nSnsDefect{7}:=1;
        ENDIF
        IF bHbltcSns08=TRUE AND DI_W07_Sns08=1 THEN
            bSnsDefect:=TRUE;
            nSnsDefect{8}:=1;
        ENDIF
        IF bHbltcSns09=TRUE AND DI_W08_Sns09=1 THEN
            bSnsDefect:=TRUE;
            nSnsDefect{9}:=1;
        ENDIF
        IF bHbltcSns10=TRUE AND DI_W09_Sns10=1 THEN
            bSnsDefect:=TRUE;
            nSnsDefect{10}:=1;
        ENDIF

        IF bSnsDefect=TRUE THEN
            USR_Print(s_LineaVuota{nIdioma});
            Reset DO_P015_PcIncompleta;
            PulseDO\PLength:=2,DO_P015_PcIncompleta;
            Reset DO_P006_AnomaliaRobo;
            PulseDO\PLength:=2,DO_P006_AnomaliaRobo;
            FOR i FROM 1 TO 10 DO
                IF nSnsDefect{i}<>0 THEN
                    USR_Print(s_GuastoFtc1{nIdioma}+NumToStr(i,0)+s_GuastoFtc2{nIdioma});
                ENDIF
            ENDFOR
            Set DO_V08_LuzVermelha;
            ROB_AlarmeAcustico(2);
            TPReadFK nKey,s_AnomaliaTestFtc{nIdioma},stEmpty,stEmpty,stEmpty,stEmpty,"OK"\DIBreak:=DI_V01_ResetAllRob\BreakFlag:=errvar;
            IF errvar=ERR_TP_DIBREAK nKey:=5;
            TEST nKey
            CASE 5:
                nKey:=0;
                GOTO check;
            ENDTEST
        ENDIF
        Reset DO_V08_LuzVermelha;
        Reset DO_P015_PcIncompleta;
        Reset DO_P006_AnomaliaRobo;

    ENDPROC

    !*********************************************************
    ! Routine:  SNS_CtrlPeca()
    !*********************************************************
    PROC SNS_CtrlPeca()

        bErrCtrlSns:=FALSE;

        ! inicializaCAO array nSnsAusentes
        FOR i FROM 1 TO 10 DO
            nSnsAusentes{i}:=0;
        ENDFOR

        ! control sesnores
        IF bHbltcSns01=TRUE AND DI_W00_Sns01=0 THEN
            bErrCtrlSns:=TRUE;
            nSnsAusentes{1}:=1;
        ENDIF
        IF bHbltcSns02=TRUE AND DI_W01_Sns02=0 THEN
            bErrCtrlSns:=TRUE;
            nSnsAusentes{2}:=1;
        ENDIF
        IF bHbltcSns03=TRUE AND DI_W02_Sns03=0 THEN
            bErrCtrlSns:=TRUE;
            nSnsAusentes{3}:=1;
        ENDIF
        IF bHbltcSns04=TRUE AND DI_W03_Sns04=0 THEN
            bErrCtrlSns:=TRUE;
            nSnsAusentes{4}:=1;
        ENDIF
        IF bHbltcSns05=TRUE AND DI_W04_Sns05=0 THEN
            bErrCtrlSns:=TRUE;
            nSnsAusentes{5}:=1;
        ENDIF
        IF bHbltcSns06=TRUE AND DI_W05_Sns06=0 THEN
            bErrCtrlSns:=TRUE;
            nSnsAusentes{6}:=1;
        ENDIF
        IF bHbltcSns07=TRUE AND DI_W06_Sns07=0 THEN
            bErrCtrlSns:=TRUE;
            nSnsAusentes{7}:=1;
        ENDIF
        IF bHbltcSns08=TRUE AND DI_W07_Sns08=0 THEN
            bErrCtrlSns:=TRUE;
            nSnsAusentes{8}:=1;
        ENDIF
        IF bHbltcSns09=TRUE AND DI_W08_Sns09=0 THEN
            bErrCtrlSns:=TRUE;
            nSnsAusentes{9}:=1;
        ENDIF
        IF bHbltcSns10=TRUE AND DI_W09_Sns10=0 THEN
            bErrCtrlSns:=TRUE;
            nSnsAusentes{10}:=1;
        ENDIF

        ! anomal?a PECA incompleta
        IF bErrCtrlSns=TRUE THEN
            Reset DO_P015_PcIncompleta;
            ! PulseDO\PLength:=2,DO_P015_PcIncompleta;
            Set DO_P015_PcIncompleta;
            Reset DO_P006_AnomaliaRobo;
            PulseDO\PLength:=2,DO_P006_AnomaliaRobo;
            FOR i FROM 1 TO 10 DO
                IF nSnsAusentes{i}<>0 THEN
                    USR_Print(s_ErroreFtc{nIdioma}+NumToStr(i,0));
                ENDIF
            ENDFOR
            Set DO_V08_LuzVermelha;
            ROB_AlarmeAcustico(2);
            USR_Print(s_AttesaReset{nIdioma});
            WaitDI DI_V01_ResetAllRob,1;
            Reset DO_V08_LuzVermelha;
            Reset DO_P015_PcIncompleta;
            Reset DO_P006_AnomaliaRobo;
        ENDIF

    ENDPROC

    !*********************************************************
    ! Routine:  MDF_Start()
    !*********************************************************
    PROC MDF_Start()
        VAR bool bStop:=FALSE;

        IF (bHbltcStopPrensaNoAuto=TRUE AND bHbltcPrensaColoc=TRUE AND DI_P309_05_HbltcPrensa=1 AND DI_P240_PrnAuto=0) THEN
            USR_Print(s_AutomaticoPrensa{nIdioma});
            bStop:=TRUE;
        ENDIF

        IF (bHbltcUtilInt=TRUE AND bHbltcSnsUtilInt=TRUE AND bHbltcStopUtilSns=TRUE AND DI_W17_SnsUtilIntermedio=1) THEN
            USR_Print(s_UtilOccupato{nIdioma});
            bStop:=TRUE;
        ENDIF

        IF bStop=TRUE THEN
            Set DO_V08_LuzVermelha;
            ROB_AlarmeAcustico(2);
            Reset DO_P006_AnomaliaRobo;
            PulseDO\PLength:=2.1,DO_P006_AnomaliaRobo;
            USR_Print(s_AttesaReset{nIdioma});
            WaitDI DI_V01_ResetAllRob,1;
            Reset DO_V08_LuzVermelha;
            Reset DO_W03_AlarmeAcustico;
            Reset DO_P006_AnomaliaRobo;
        ENDIF
        !
        IF bPcIncompleta=FALSE THEN
            Reset DO_P013_OkFecharMdf;
            PulseDO\PLength:=1,DO_P013_OkFecharMdf;
        ENDIF

        IF DI_P016_MdfFimCiclo=1 THEN
            ROB_AlarmeAcustico(2);
            USR_Print(s_FineCiclo{nIdioma});
        ENDIF

        Incr ROB_nPcTotal;
        IF (bPcBoaDeMdf=TRUE AND bPcIncompleta=FALSE) THEN
            Incr ROB_nPcBuona;
        ELSE
            Incr ROB_nPcRejeicao;
        ENDIF

        ClkReset timerROB;
        ClkStart timerROB;

    ENDPROC

